# B&R Automation Studio project Y4_V3_1 (part 8)

#### S_Page13.st - Cyclic code
```iecst
(********************************************************************
 * COPYRIGHT --
 ********************************************************************
 * Program: S_Page13
 * File: S_Page13.st
 * Author: nicke
 * Created: May 02, 2013
 ********************************************************************
 * Implementation of program S_Page13
 ********************************************************************)

PROGRAM _CYCLIC

	//SETTINGS SCREEN
	ServiceVis.P13.EnableIndex	:=	LIMIT(0,ServiceVis.P13.EnableIndex,24)	;
	ServiceVis.P13.Status[0]	:=	HIDE	;
	ServiceVis.P13.Status[1]	:=	HIDE	;
	ServiceVis.P13.Status[2]	:=	HIDE	;
	ServiceVis.P13.Status[3]	:=	HIDE	;
	ServiceVis.P13.Status[4]	:=	HIDE	;
	ServiceVis.P13.Status[5]	:=	HIDE	;
	ServiceVis.P13.Status[6]	:=	HIDE	;
	ServiceVis.P13.Status[7]	:=	HIDE	;
	ServiceVis.P13.Status[8]	:=	HIDE	;
	ServiceVis.P13.Status[9]	:=	HIDE	;
	ServiceVis.P13.Status[10]	:=	HIDE	;
	ServiceVis.P13.Colour[1]	:=	BLUE	;
	ServiceVis.P13.Colour[2]	:=	BLUE	;
	ServiceVis.P13.Colour[3]	:=	BLUE	;
	ServiceVis.P13.Colour[4]	:=	BLUE	;
	ServiceVis.P13.Colour[5]	:=	BLUE	;
	ServiceVis.P13.Colour[6]	:=	BLUE	;

	CASE ServiceVis.P13.EnableIndex OF
		0:
			ServiceVis.P13.Status[0]	:=	SHOW	;
			ServiceVis.CalcBelt.Disp	:=	HIDE	;
		1:
			ServiceVis.P13.Status[1]	:=	SHOW	;
			ServiceVis.P13.Status[9]	:=	SHOW	;
			ServiceVis.P13.Colour[1]	:=	BLUE_ACTIVE	;
		2:
			ServiceVis.P13.Status[2]	:=	SHOW	;
			ServiceVis.P13.Status[9]	:=	SHOW	;
			ServiceVis.P13.Colour[2]	:=	BLUE_ACTIVE	;
			ServiceVis.CalcBelt.Disp	:=	HIDE	;
		3:
			ServiceVis.P13.Status[3]	:=	SHOW	;
			ServiceVis.P13.Status[9]	:=	SHOW	;
			ServiceVis.P13.Colour[3]	:=	BLUE_ACTIVE	;
			ServiceVis.CalcBelt.Disp	:=	HIDE	;
		4:
			ServiceVis.P13.Status[4]	:=	SHOW	;
			ServiceVis.P13.Status[9]	:=	SHOW	;
			ServiceVis.P13.Colour[4]	:=	BLUE_ACTIVE	;
			ServiceVis.CalcBelt.Disp	:=	HIDE	;
		5:
			ServiceVis.P13.Status[5]	:=	SHOW	;
			ServiceVis.P13.Status[9]	:=	SHOW	;
			ServiceVis.P13.Colour[5]	:=	BLUE_ACTIVE	;
			ServiceVis.CalcBelt.Disp	:=	HIDE	;
		6:
			ServiceVis.P13.Status[6]	:=	SHOW	;
			ServiceVis.P13.Status[9]	:=	SHOW	;
			ServiceVis.P13.Colour[6]	:=	BLUE_ACTIVE	;
			ServiceVis.CalcBelt.Disp	:=	HIDE	;
		7:
			ServiceVis.P13.Status[7]	:=	SHOW	;
			ServiceVis.CalcBelt.Disp	:=	HIDE	;
		8:
			ServiceVis.P13.Status[8]	:=	SHOW	;
			ServiceVis.P13.Status[3]	:=	SHOW	;
			ServiceVis.P13.Status[9]	:=	SHOW	;
			ServiceVis.P13.Colour[3]	:=	BLUE_ACTIVE	;
			ServiceVis.CalcBelt.Disp	:=	HIDE	;
		10:
			ServiceVis.P13.Status[10]	:=	SHOW	;
			ServiceVis.P13.Status[6]	:=	SHOW	;
			ServiceVis.P13.Status[9]	:=	SHOW	;
			ServiceVis.P13.Colour[6]	:=	BLUE_ACTIVE	;
			ServiceVis.CalcBelt.Disp	:=	HIDE	;

	END_CASE

	//CALCULATE WHEN LAYER HAS CHANGED
	ServiceVis.P13.Changed	:=	FALSE	;
	ServiceVis.P13.New	:=	ServiceVis.P13.EnableIndex	;
	IF(ServiceVis.P13.New <> ServiceVis.P13.Old) THEN
		ServiceVis.P13.Changed	:=	TRUE	;
	END_IF
	IF EDGEPOS(ServiceVis.P13.Changed) THEN
		ServiceVis.P13Delays.EnableIndex	:=	24	;
		ServiceVis.P13Servos.EnableIndex	:=	24	;
		ServiceVis.P13System.EnableIndex	:=	24	;
		ServiceVis.P13Timeouts.EnableIndex	:=	24	;
		ServiceVis.P13Help1.EnableIndex	:=	24	;
		ServiceVis.P13Help2.EnableIndex	:=	24	;
	END_IF
	ServiceVis.P13.Old	:=	ServiceVis.P13.EnableIndex	;

	//SETTINGS DELAYS SCREEN
	ServiceVis.P13Delays.Status[0]	:=	HIDE	;
	ServiceVis.P13Delays.Status[1]	:=	HIDE	;
	ServiceVis.P13Delays.Status[2]	:=	HIDE	;
	ServiceVis.P13Delays.Status[3]	:=	HIDE	;
	ServiceVis.P13Delays.Status[4]	:=	HIDE	;
	ServiceVis.P13Delays.Status[5]	:=	HIDE	;
	ServiceVis.P13Delays.Status[6]	:=	HIDE	;
	ServiceVis.P13Delays.Status[7]	:=	HIDE	;
	ServiceVis.P13Delays.Status[8]	:=	HIDE	;
	ServiceVis.P13Delays.Status[9]	:=	HIDE	;
	ServiceVis.P13Delays.Status[10]	:=	HIDE	;
	ServiceVis.P13Delays.Colour[0]	:=	BLUE	;
	ServiceVis.P13Delays.Colour[1]	:=	BLUE	;
	ServiceVis.P13Delays.Colour[2]	:=	BLUE	;
	ServiceVis.P13Delays.Colour[3]	:=	BLUE	;
	ServiceVis.P13Delays.Colour[4]	:=	BLUE	;
	ServiceVis.P13Delays.Colour[5]	:=	BLUE	;
	ServiceVis.P13Delays.Colour[6]	:=	BLUE	;
	ServiceVis.P13Delays.Colour[7]	:=	BLUE	;
	ServiceVis.P13Delays.Colour[8]	:=	BLUE	;

	CASE ServiceVis.P13Delays.EnableIndex OF
		0..8://LayerDelay[1..9]
			ServiceVis.P13Delays.Status[ServiceVis.P13Delays.EnableIndex]	:=	SHOW	;
			ServiceVis.P13Delays.Colour[ServiceVis.P13Delays.EnableIndex]	:=	BLUE_ACTIVE	;
			ServiceVis.P13Delays.Status[9]	:=	SHOW	;//LayerDelays
			ServiceVis.P13.Status[1]	:=	HIDE	;//Layer2
			ServiceVis.P13.Status[9]	:=	HIDE	;//Layers
		10:
			ServiceVis.P13Delays.Status[10]	:=	SHOW	;
	END_CASE

	CASE ServiceVis.P13Delays.EnableIndex OF
		0,2,4,5,6,7,8,24:
			ServiceVis.CalcBelt.Disp	:=	HIDE	;
	END_CASE

	//CALCULATE WHEN LAYER HAS CHANGED
	ServiceVis.P13Delays.Changed	:=	FALSE	;
	ServiceVis.P13Delays.New	:=	ServiceVis.P13Delays.EnableIndex	;
	IF(ServiceVis.P13Delays.New <> ServiceVis.P13Delays.Old) THEN
		ServiceVis.P13Delays.Changed	:=	TRUE	;
	END_IF
	IF EDGEPOS(ServiceVis.P13Delays.Changed) THEN
		ServiceVis.P13Help1.EnableIndex	:=	24	;
		ServiceVis.P13Help2.EnableIndex	:=	24	;
	END_IF
	ServiceVis.P13Delays.Old	:=	ServiceVis.P13Delays.EnableIndex	;

	//CALCULATOR FOR BELT DISPLAY
	IF (ServiceVis.CalcBelt.Disp = SHOW) THEN
		IF (ServiceVis.CalcBelt.Delay) THEN
			ServiceVis.CalcBelt.Adjust	:= 	1 - ((ServiceVis.CalcBelt.Unground + 300)/(Speeds.SpeedSeam/6))	;
		ELSE
			ServiceVis.CalcBelt.Adjust	:= 	(ServiceVis.CalcBelt.Unground + 300)/(Speeds.SpeedSeam/6);
		END_IF
		ServiceVis.CalcBelt.New	:= 	(ServiceVis.CalcBelt.Current + ServiceVis.CalcBelt.Adjust)	;

		IF (ServiceVis.CalcBelt.Unground = 0) THEN
			ServiceVis.CalcBelt.Adjust	:= 	0	;
			ServiceVis.CalcBelt.New	:= 	0	;
		END_IF
	END_IF

	//SETTINGS DRIVES SCREEN
	ServiceVis.P13Drives.Status[0]	:=	HIDE	;
	ServiceVis.P13Drives.Status[1]	:=	HIDE	;
	ServiceVis.P13Drives.Status[2]	:=	HIDE	;
	ServiceVis.P13Drives.Status[3]	:=	HIDE	;
	ServiceVis.P13Drives.Status[4]	:=	HIDE	;
	ServiceVis.P13Drives.Status[5]	:=	HIDE	;
	ServiceVis.P13Drives.Status[6]	:=	HIDE	;
	ServiceVis.P13Drives.Status[7]	:=	HIDE	;
	ServiceVis.P13Drives.Status[8]	:=	HIDE	;
	ServiceVis.P13Drives.Status[9]	:=	HIDE	;
	ServiceVis.P13Drives.Status[10]:=	HIDE	;
	ServiceVis.P13Drives.Status[11]:=	HIDE	;
	ServiceVis.P13Drives.Status[12]:=	HIDE	;
	ServiceVis.P13Drives.Status[13]:=	HIDE	;
	ServiceVis.P13Drives.Status[14]:=	HIDE	;
	ServiceVis.P13Drives.Status[15]:=	HIDE	;
	ServiceVis.P13Drives.Status[20]:=	HIDE	;
	ServiceVis.P13Drives.Status[21]:=	HIDE	;
	ServiceVis.P13Drives.Status[22]:=	HIDE	;
	ServiceVis.P13Drives.Colour[0]	:=	BLUE	;
	ServiceVis.P13Drives.Colour[1]	:=	BLUE	;
	ServiceVis.P13Drives.Colour[2]	:=	BLUE	;
	ServiceVis.P13Drives.Colour[3]	:=	BLUE	;
	ServiceVis.P13Drives.Colour[4]	:=	BLUE	;
	ServiceVis.P13Drives.Colour[5]	:=	BLUE	;
	ServiceVis.P13Drives.Colour[6]	:=	BLUE	;

	CASE ServiceVis.P13Drives.EnableIndex OF
		0..6:
			ServiceVis.P13Drives.Status[ServiceVis.P13Drives.EnableIndex]	:=	SHOW	;
			ServiceVis.P13Drives.Colour[ServiceVis.P13Drives.EnableIndex]	:=	BLUE_ACTIVE	;
			ServiceVis.P13Drives.Status[9]	:=	SHOW	;
			ServiceVis.P13.Status[2]	:=	HIDE	;
			ServiceVis.P13.Status[9]	:=	HIDE	;
			IF(ServiceLevel.Level > SUPERVISOR) THEN
				ServiceVis.P13Drives.Status[ServiceVis.P13Drives.EnableIndex + 9]	:=	SHOW	;
			END_IF
		7:
			ServiceVis.P13Drives.Status[7]	:=	SHOW	;
		8:
			ServiceVis.P13Drives.Status[8]	:=	SHOW	;
	END_CASE

	//CALCULATE WHEN LAYER HAS CHANGED
	ServiceVis.P13Drives.Changed	:=	FALSE	;
	ServiceVis.P13Drives.New	:=	ServiceVis.P13Drives.EnableIndex	;
	IF(ServiceVis.P13Drives.New <> ServiceVis.P13Drives.Old) THEN
		ServiceVis.P13Drives.Changed	:=	TRUE	;
	END_IF
	IF EDGEPOS(ServiceVis.P13Drives.Changed) THEN
		ServiceVis.P13Help1.EnableIndex	:=	24	;
		ServiceVis.P13Help2.EnableIndex	:=	24	;
	END_IF
	ServiceVis.P13Drives.Old	:=	ServiceVis.P13Drives.EnableIndex	;

	//HIGHLIGHT SELECTED BATCHING MODE COLOUR
	CASE InvPerms.CLB.Analog OF
		NO_ANALOG:
			ServiceVis.P13.Colour[7]	:=	WHITE			;
			ServiceVis.P13.Colour[8]	:=	DROP_UNSELECTED	;
			ServiceVis.P13.Colour[9]	:=	DROP_UNSELECTED	;
			ServiceVis.P13.Colour[10]	:=	DROP_UNSELECTED	;
			ServiceVis.P13.Colour[11]	:=	DROP_UNSELECTED	;
		VOLTAGE_TYPE_1:
			ServiceVis.P13.Colour[7]	:=	DROP_UNSELECTED	;
			ServiceVis.P13.Colour[8]	:=	WHITE			;
			ServiceVis.P13.Colour[9]	:=	DROP_UNSELECTED	;
			ServiceVis.P13.Colour[10]	:=	DROP_UNSELECTED	;
			ServiceVis.P13.Colour[11]	:=	DROP_UNSELECTED	;
		CURRENT_TYPE_1:
			ServiceVis.P13.Colour[7]	:=	DROP_UNSELECTED	;
			ServiceVis.P13.Colour[8]	:=	DROP_UNSELECTED	;
			ServiceVis.P13.Colour[9]	:=	DROP_UNSELECTED	;
			ServiceVis.P13.Colour[10]	:=	WHITE			;
			ServiceVis.P13.Colour[11]	:=	DROP_UNSELECTED	;
		CURRENT_TYPE_2:
			ServiceVis.P13.Colour[7]	:=	DROP_UNSELECTED	;
			ServiceVis.P13.Colour[8]	:=	DROP_UNSELECTED	;
			ServiceVis.P13.Colour[9]	:=	DROP_UNSELECTED	;
			ServiceVis.P13.Colour[10]	:=	DROP_UNSELECTED	;
			ServiceVis.P13.Colour[11]	:=	WHITE			;
	END_CASE

	//SETTINGS SERVOS SCREEN
	ServiceVis.P13Servos.Status[0]	:=	HIDE	;
	ServiceVis.P13Servos.Status[1]	:=	HIDE	;
	ServiceVis.P13Servos.Status[2]	:=	HIDE	;
	ServiceVis.P13Servos.Status[3]	:=	HIDE	;
	ServiceVis.P13Servos.Status[4]	:=	HIDE	;
	ServiceVis.P13Servos.Status[5]	:=	HIDE	;
	ServiceVis.P13Servos.Status[6]	:=	HIDE	;
	ServiceVis.P13Servos.Status[7]	:=	HIDE	;
	ServiceVis.P13Servos.Status[8]	:=	HIDE	;
	ServiceVis.P13Servos.Status[9]	:=	HIDE	;
	ServiceVis.P13Servos.Colour[0]	:=	BLUE	;
	ServiceVis.P13Servos.Colour[1]	:=	BLUE	;
	ServiceVis.P13Servos.Colour[2]	:=	BLUE	;
	ServiceVis.P13Servos.Colour[3]	:=	BLUE	;
	ServiceVis.P13Servos.Colour[4]	:=	BLUE	;
	ServiceVis.P13Servos.Colour[5]	:=	BLUE	;
	ServiceVis.P13Servos.Colour[6]	:=	BLUE	;

	CASE ServiceVis.P13Servos.EnableIndex OF
		0..6:
			ServiceVis.P13Servos.Status[ServiceVis.P13Servos.EnableIndex]	:=	SHOW	;
			ServiceVis.P13Servos.Colour[ServiceVis.P13Servos.EnableIndex]	:=	BLUE_ACTIVE	;
			ServiceVis.P13Servos.Status[9]	:=	SHOW	;
			ServiceVis.P13.Status[2]	:=	HIDE	;
			ServiceVis.P13.Status[9]	:=	HIDE	;
		7:
			ServiceVis.P13Servos.Status[7]	:=	SHOW	;
		8:
			ServiceVis.P13Servos.Status[8]	:=	SHOW	;
	END_CASE

	//CALCULATE WHEN LAYER HAS CHANGED
	ServiceVis.P13Servos.Changed	:=	FALSE	;
	ServiceVis.P13Servos.New	:=	ServiceVis.P13Servos.EnableIndex	;
	IF(ServiceVis.P13Servos.New <> ServiceVis.P13Servos.Old) THEN
		ServiceVis.P13Servos.Changed	:=	TRUE	;
	END_IF
	IF EDGEPOS(ServiceVis.P13Servos.Changed) THEN
		ServiceVis.P13Help1.EnableIndex	:=	24	;
		ServiceVis.P13Help2.EnableIndex	:=	24	;
	END_IF
	ServiceVis.P13Servos.Old	:=	ServiceVis.P13Servos.EnableIndex	;

	//SETTINGS SYSTEM SCREEN
	ServiceVis.P13System.Status[0]	:=	HIDE	;
	ServiceVis.P13System.Status[1]	:=	HIDE	;
	ServiceVis.P13System.Status[2]	:=	HIDE	;
	ServiceVis.P13System.Status[3]	:=	HIDE	;
	ServiceVis.P13System.Status[4]	:=	HIDE	;
	ServiceVis.P13System.Status[5]	:=	HIDE	;
	ServiceVis.P13System.Status[6]	:=	HIDE	;
	ServiceVis.P13System.Status[7]	:=	HIDE	;
	ServiceVis.P13System.Status[8]	:=	HIDE	;
	ServiceVis.P13System.Status[9]	:=	HIDE	;
	ServiceVis.P13System.Colour[0]	:=	BLUE	;
	ServiceVis.P13System.Colour[1]	:=	BLUE	;
	ServiceVis.P13System.Colour[2]	:=	BLUE	;
	ServiceVis.P13System.Colour[3]	:=	BLUE	;
	ServiceVis.P13System.Colour[4]	:=	BLUE	;
	ServiceVis.P13System.Colour[5]	:=	BLUE	;
	ServiceVis.P13System.Colour[6]	:=	BLUE	;

	CASE ServiceVis.P13System.EnableIndex OF
		0..6:
			ServiceVis.P13System.Status[ServiceVis.P13System.EnableIndex]	:=	SHOW	;
			ServiceVis.P13System.Colour[ServiceVis.P13System.EnableIndex]	:=	BLUE_ACTIVE	;
			ServiceVis.P13System.Status[9]	:=	SHOW	;
			ServiceVis.P13.Status[4]	:=	HIDE	;
			ServiceVis.P13.Status[9]	:=	HIDE	;
		7:
			ServiceVis.P13System.Status[7]	:=	SHOW	;
		8:
			ServiceVis.P13System.Status[8]	:=	SHOW	;
	END_CASE

	//CALCULATE WHEN LAYER HAS CHANGED
	ServiceVis.P13System.Changed	:=	FALSE	;
	ServiceVis.P13System.New	:=	ServiceVis.P13System.EnableIndex	;
	IF(ServiceVis.P13System.New <> ServiceVis.P13System.Old) THEN
		ServiceVis.P13System.Changed	:=	TRUE	;
	END_IF
	IF EDGEPOS(ServiceVis.P13System.Changed) THEN
		ServiceVis.P13Help1.EnableIndex	:=	24	;
		ServiceVis.P13Help2.EnableIndex	:=	24	;
	END_IF
	ServiceVis.P13System.Old	:=	ServiceVis.P13System.EnableIndex	;

	//SETTINGS TIMEOUT SCREEN
	ServiceVis.P13Timeouts.Status[0]	:=	HIDE	;
	ServiceVis.P13Timeouts.Status[1]	:=	HIDE	;
	ServiceVis.P13Timeouts.Status[2]	:=	HIDE	;
	ServiceVis.P13Timeouts.Status[3]	:=	HIDE	;
	ServiceVis.P13Timeouts.Status[4]	:=	HIDE	;
	ServiceVis.P13Timeouts.Status[5]	:=	HIDE	;
	ServiceVis.P13Timeouts.Status[6]	:=	HIDE	;
	ServiceVis.P13Timeouts.Status[7]	:=	HIDE	;
	ServiceVis.P13Timeouts.Status[8]	:=	HIDE	;
	ServiceVis.P13Timeouts.Status[9]	:=	HIDE	;
	ServiceVis.P13Timeouts.Colour[0]	:=	BLUE	;
	ServiceVis.P13Timeouts.Colour[1]	:=	BLUE	;
	ServiceVis.P13Timeouts.Colour[2]	:=	BLUE	;
	ServiceVis.P13Timeouts.Colour[3]	:=	BLUE	;
	ServiceVis.P13Timeouts.Colour[4]	:=	BLUE	;
	ServiceVis.P13Timeouts.Colour[5]	:=	BLUE	;
	ServiceVis.P13Timeouts.Colour[6]	:=	BLUE	;

	CASE ServiceVis.P13Timeouts.EnableIndex OF
		0..6:
			ServiceVis.P13Timeouts.Status[ServiceVis.P13Timeouts.EnableIndex]	:=	SHOW	;
			ServiceVis.P13Timeouts.Colour[ServiceVis.P13Timeouts.EnableIndex]	:=	BLUE_ACTIVE	;
			ServiceVis.P13Timeouts.Status[9]	:=	SHOW	;
			ServiceVis.P13.Status[5]	:=	HIDE	;
			ServiceVis.P13.Status[9]	:=	HIDE	;
		7:
			ServiceVis.P13Timeouts.Status[7]	:=	SHOW	;
		8:
			ServiceVis.P13Timeouts.Status[8]	:=	SHOW	;
	END_CASE

	//CALCULATE WHEN LAYER HAS CHANGED
	ServiceVis.P13Timeouts.Changed	:=	FALSE	;
	ServiceVis.P13Timeouts.New	:=	ServiceVis.P13Timeouts.EnableIndex	;
	IF(ServiceVis.P13Timeouts.New <> ServiceVis.P13Timeouts.Old) THEN
		ServiceVis.P13Timeouts.Changed	:=	TRUE	;
	END_IF
	IF EDGEPOS(ServiceVis.P13Timeouts.Changed) THEN
		ServiceVis.P13Help1.EnableIndex	:=	24	;
		ServiceVis.P13Help2.EnableIndex	:=	24	;
	END_IF
	ServiceVis.P13Timeouts.Old	:=	ServiceVis.P13Timeouts.EnableIndex	;

	//HELP LAYERS CONTROL
	memcpy(ADR(ServiceVis.P13Help1.Status),ADR(ServiceVis.HideAll),SIZEOF(ServiceVis.HideAll));
	ServiceVis.P13Help1.Colour[0]	:=	BLUE	;
	ServiceVis.P13Help1.Colour[1]	:=	BLUE	;
	ServiceVis.P13Help1.Colour[2]	:=	BLUE	;
	ServiceVis.P13Help1.Colour[3]	:=	BLUE	;
	ServiceVis.P13Help1.Colour[4]	:=	BLUE	;
	ServiceVis.P13Help1.Colour[5]	:=	BLUE	;
	ServiceVis.P13Help1.Colour[6]	:=	BLUE	;
	ServiceVis.P13Help1.Colour[7]	:=	BLUE	;
	ServiceVis.P13Help1.Colour[8]	:=	BLUE	;
	ServiceVis.P13Help1.Colour[9]	:=	BLUE	;

	CASE ServiceVis.P13Help1.EnableIndex OF
		0..23:
			ServiceVis.P13Help1.Status[ServiceVis.P13Help1.EnableIndex]	:=	SHOW	;
		24:
			ServiceVis.P13Help1.Index	:=	0	;
	END_CASE

	CASE ServiceVis.P13Help1.Index OF
		0..9:
			ServiceVis.P13Help1.Colour[ServiceVis.P13Help1.Index]	:=	BLUE_ACTIVE	;
	END_CASE

	//HELP LAYERS CONTROL 2
	memcpy(ADR(ServiceVis.P13Help2.Status),ADR(ServiceVis.HideAll),SIZEOF(ServiceVis.HideAll));
	ServiceVis.P13Help2.Colour[0]	:=	BLUE	;
	ServiceVis.P13Help2.Colour[1]	:=	BLUE	;
	ServiceVis.P13Help2.Colour[2]	:=	BLUE	;
	ServiceVis.P13Help2.Colour[3]	:=	BLUE	;
	ServiceVis.P13Help2.Colour[4]	:=	BLUE	;
	ServiceVis.P13Help2.Colour[5]	:=	BLUE	;
	ServiceVis.P13Help2.Colour[6]	:=	BLUE	;
	ServiceVis.P13Help2.Colour[7]	:=	BLUE	;
	ServiceVis.P13Help2.Colour[8]	:=	BLUE	;
	ServiceVis.P13Help2.Colour[9]	:=	BLUE	;
	ServiceVis.P13Help2.Colour[10]	:=	BLUE	;

	CASE ServiceVis.P13Help2.EnableIndex OF
		0..23:
			ServiceVis.P13Help2.Status[ServiceVis.P13Help2.EnableIndex]	:=	SHOW	;
		24:
			ServiceVis.P13Help2.Index	:=	0	;
	END_CASE

	CASE ServiceVis.P13Help2.Index OF
		0..10:
			ServiceVis.P13Help2.Colour[ServiceVis.P13Help2.Index]	:=	BLUE_ACTIVE	;
	END_CASE

END_PROGRAM
```

### Program Logical/VisControl/ServiceControl/S_Page14 (IEC) - Drives screen control

#### S_Page14.st - Cyclic code
```iecst
(********************************************************************
 * COPYRIGHT --
 ********************************************************************
 * Program: S_Page14
 * File: S_Page14.st
 * Author: nicke
 * Created: May 02, 2013
 ********************************************************************
 * Implementation of program S_Page14
 ********************************************************************)

PROGRAM _CYCLIC

	//DRIVES SCREEN
	memcpy(ADR(ServiceVis.P14.Status),ADR(ServiceVis.HideAll),SIZEOF(ServiceVis.HideAll));
	ServiceVis.P14.Colour[0]	:=	VIOLET	;
	ServiceVis.P14.Colour[1]	:=	VIOLET	;
	ServiceVis.P14.Colour[2]	:=	VIOLET	;
	ServiceVis.P14.Colour[3]	:=	VIOLET	;
	ServiceVis.P14.Colour[4]	:=	VIOLET	;
	ServiceVis.P14.Colour[5]	:=	VIOLET	;
	ServiceVis.P14.Colour[6]	:=	VIOLET	;

	CASE ServiceVis.P14.EnableIndex OF
		0..6:
			ServiceVis.P14.Status[ServiceVis.P14.EnableIndex]	:=	SHOW	;
			ServiceVis.P14.Colour[ServiceVis.P14.EnableIndex]	:=	VIOLET_ACTIVE	;
	END_CASE

	IF (Control.Achieved1) OR(Control.Test) THEN
		ServiceVis.P14.Status[8]	:=	SHOW	;
	END_IF

	IF(Control.Test) THEN
		ServiceVis.P14.Status[9]	:=	SHOW	;
	END_IF

	//CALCULATE WHEN LAYER HAS CHANGED
	ServiceVis.P14.Changed	:=	FALSE	;
	ServiceVis.P14.New	:=	ServiceVis.P14.EnableIndex	;
	IF(ServiceVis.P14.New <> ServiceVis.P14.Old) THEN
		ServiceVis.P14.Changed	:=	TRUE	;
	END_IF
	IF EDGEPOS(ServiceVis.P14.Changed) THEN
		ServiceVis.P14Layer.EnableIndex		:=	24	;
		ServiceVis.P14Status.EnableIndex	:=	24	;
		ServiceVis.P14Help.EnableIndex		:=	24	;
	END_IF
	ServiceVis.P14.Old	:=	ServiceVis.P14.EnableIndex	;

	memcpy(ADR(ServiceVis.P14Layer.Status),ADR(ServiceVis.HideAll),SIZEOF(ServiceVis.HideAll));

	CASE ServiceVis.P14Layer.EnableIndex OF
		0..19:
			ServiceVis.P14Layer.Status[ServiceVis.P14Layer.EnableIndex]	:=	SHOW	;
	END_CASE

END_PROGRAM
```

### Program Logical/VisControl/ServiceControl/S_Page15 (IEC) - Servo screen control

#### S_Page15.st - Cyclic code
```iecst
(********************************************************************
 * COPYRIGHT --
 ********************************************************************
 * Program: S_Page15
 * File: S_Page15.st
 * Author: nicke
 * Created: May 02, 2013
 ********************************************************************
 * Implementation of program S_Page15
 ********************************************************************)

PROGRAM _CYCLIC

	//SERVOS SCREEN
	memcpy(ADR(ServiceVis.P15.Status),ADR(ServiceVis.HideAll),SIZEOF(ServiceVis.HideAll));
	ServiceVis.P15.Colour[0]	:=	GREEN1	;
	ServiceVis.P15.Colour[1]	:=	GREEN1	;
	ServiceVis.P15.Colour[2]	:=	GREEN1	;
	ServiceVis.P15.Colour[3]	:=	GREEN1	;
	ServiceVis.P15.Colour[4]	:=	GREEN1	;
	ServiceVis.P15.Colour[5]	:=	GREEN1	;
	ServiceVis.P15.Colour[6]	:=	GREEN1	;

	CASE ServiceVis.P15.EnableIndex OF
		0..6:
			ServiceVis.P15.Status[ServiceVis.P15.EnableIndex]	:=	SHOW	;
			ServiceVis.P15.Colour[ServiceVis.P15.EnableIndex]	:=	GREEN1_ACTIVE	;
	END_CASE

	IF(Control.Test) THEN
		ServiceVis.P15.Status[8]	:=	SHOW	;
		//	ELSE
		//		ServiceVis.P15Layer.EnableIndex	:=	24	;
	END_IF

	//CALCULATE WHEN LAYER HAS CHANGED
	ServiceVis.P15.Changed	:=	FALSE	;
	ServiceVis.P15.New	:=	ServiceVis.P15.EnableIndex	;
	IF(ServiceVis.P15.New <> ServiceVis.P15.Old) THEN
		ServiceVis.P15.Changed	:=	TRUE	;
	END_IF
	IF EDGEPOS(ServiceVis.P15.Changed) THEN
		ServiceVis.P15Layer.EnableIndex	:=	24	;
	END_IF
	ServiceVis.P15.Old	:=	ServiceVis.P15.EnableIndex	;

	memcpy(ADR(ServiceVis.P15Layer.Status),ADR(ServiceVis.HideAll),SIZEOF(ServiceVis.HideAll));

	CASE ServiceVis.P15Layer.EnableIndex OF
		0..15:
			ServiceVis.P15Layer.Status[ServiceVis.P15Layer.EnableIndex]	:=	SHOW	;
	END_CASE

	IF(Control.Test) THEN
	ELSE
		ServiceVis.P15Layer.Status[0]	:=	HIDE	;
		ServiceVis.P15Layer.Status[1]	:=	HIDE	;
		ServiceVis.P15Layer.Status[2]	:=	HIDE	;
	END_IF

END_PROGRAM
```

### Program Logical/VisControl/ServiceControl/S_Page16 (IEC) - Remote screen control

#### S_Page16.st - Cyclic code
```iecst
(********************************************************************
 * COPYRIGHT --
 ********************************************************************
 * Program: S_Page16
 * File: S_Page16.st
 * Author: nicke
 * Created: May 02, 2013
 ********************************************************************
 * Implementation of program S_Page16
 ********************************************************************)

PROGRAM _CYCLIC

	//REMOTE SCREEN
	memcpy(ADR(ServiceVis.P16.Status),ADR(ServiceVis.HideAll),SIZEOF(ServiceVis.HideAll));
	ServiceVis.P16.Colour[0]	:=	LIGHTBLUE	;
	ServiceVis.P16.Colour[1]	:=	LIGHTBLUE	;
	ServiceVis.P16.Colour[2]	:=	LIGHTBLUE	;
	ServiceVis.P16.Colour[3]	:=	LIGHTBLUE	;
	ServiceVis.P16.Colour[4]	:=	LIGHTBLUE	;
	ServiceVis.P16.Colour[5]	:=	LIGHTBLUE	;
	ServiceVis.P16.Colour[6]	:=	LIGHTBLUE	;
	ServiceVis.P16.Colour[7]	:=	LIGHTBLUE	;
	ServiceVis.P16.Colour[8]	:=	LIGHTBLUE	;
	ServiceVis.P16.Colour[9]	:=	LIGHTBLUE	;
	ServiceVis.P16.Colour[10]	:=	LIGHTBLUE	;

	CASE ServiceVis.P16.EnableIndex OF
		0..7,9,10:
			ServiceVis.P16.Status[ServiceVis.P16.EnableIndex]	:=	SHOW	;
			ServiceVis.P16.Colour[ServiceVis.P16.EnableIndex]	:=	LIGHTBLUE_ACTIVE	;
	END_CASE

	IF(Control.Test) THEN
		ServiceVis.P16.Status[8]	:=	SHOW	;
	ELSE
		ServiceVis.P16.EnableIndex	:= LIMIT(0, ServiceVis.P16.EnableIndex, 6);
	END_IF

	//CALCULATE WHEN LAYER HAS CHANGED
	ServiceVis.P16.Changed	:=	FALSE	;
	ServiceVis.P16.New	:=	ServiceVis.P16.EnableIndex	;
	IF(ServiceVis.P16.New <> ServiceVis.P16.Old) THEN
		ServiceVis.P16.Changed	:=	TRUE	;
	END_IF
	IF EDGEPOS(ServiceVis.P16.Changed) THEN
		ServiceVis.P16Layer.EnableIndex	:=	24	;
	END_IF
	ServiceVis.P16.Old	:=	ServiceVis.P16.EnableIndex	;

	memcpy(ADR(ServiceVis.P16Layer.Status),ADR(ServiceVis.HideAll),SIZEOF(ServiceVis.HideAll));

	CASE ServiceVis.P16Layer.EnableIndex OF
		0..15:
			ServiceVis.P16Layer.Status[ServiceVis.P16Layer.EnableIndex]	:=	SHOW	;
	END_CASE

END_PROGRAM
```

### Program Logical/VisControl/ServiceControl/S_Page18 (IEC) - Warning screen control

#### S_Page18.st - Cyclic code
```iecst
(********************************************************************
 * COPYRIGHT --
 ********************************************************************
 * Program: S_Page18
 * File: S_Page18.st
 * Author: nicke
 * Created: May 02, 2013
 ********************************************************************
 * Implementation of program S_Page18
 ********************************************************************)

PROGRAM _CYCLIC

(* Section to control pop up warnings for flip arms *)
(*Seamer 1 Down *)
	ServiceVis.FlipDisp1.Runtime1	:=	HIDE	;
	ServiceVis.FlipDisp1.Runtime2	:=	HIDE	;
	ServiceVis.FlipDisp1.Runtime3	:=	HIDE	;
	ServiceVis.FlipDisp1.Runtime4	:=	HIDE	;

	IF ((Ax1.Active) OR NOT(Ax1.OriginSet)) AND NOT(Ax1.Block) AND(Control.Achieved1) THEN
		ServiceVis.FlipDisp1.Runtime1	:=	SHOW	;
		ServiceVis.FlipDisp1.TextIndex1	:=	BOOL_TO_USINT(NOT(S100Reed.In))	;
		ServiceVis.FlipDisp1.TextIndex2	:=	BOOL_TO_USINT(NOT(S102Reed.In))	;
		ServiceVis.FlipDisp1.TextIndex3	:=	BOOL_TO_USINT(NOT(S104Reed.In))	;
		ServiceVis.FlipDisp1.TextIndex4	:=	BOOL_TO_USINT(NOT(S106Reed.In))	;
		ServiceVis.FlipDisp1.TextIndex5	:=	BOOL_TO_USINT(NOT(S108Reed.In))	;
		ServiceVis.FlipDisp1.TextIndex6	:=	BOOL_TO_USINT(NOT(S110Reed.In))	;
		ServiceVis.FlipDisp1.TextIndex7	:=	BOOL_TO_USINT(NOT(S112Reed.In))	;
		ServiceVis.FlipDisp1.TextIndex8	:=	BOOL_TO_USINT(NOT(S114Reed.In))	;
		ServiceVis.FlipDisp1.TextIndex9	:=	BOOL_TO_USINT(NOT(S116Reed.In))	;
		ServiceVis.FlipDisp1.TextIndex10	:=	BOOL_TO_USINT(NOT(S118Reed.In))	;
		CASE Perms.FLIPARMS1 OF
			3:
				ServiceVis.FlipDisp1.Runtime2		:=	SHOW	;
			4:
				ServiceVis.FlipDisp1.Runtime2		:=	SHOW	;
				ServiceVis.FlipDisp1.Runtime3		:=	SHOW	;
			5:
				ServiceVis.FlipDisp1.Runtime2		:=	SHOW	;
				ServiceVis.FlipDisp1.Runtime3		:=	SHOW	;
				ServiceVis.FlipDisp1.Runtime4		:=	SHOW	;
		END_CASE
	END_IF

	(* Seamer 1 Up *)
	ServiceVis.FlipDisp1.Runtime5	:= HIDE	;
	ServiceVis.FlipDisp1.Runtime6	:= HIDE	;
	ServiceVis.FlipDisp1.Runtime7	:= HIDE	;
	ServiceVis.FlipDisp1.Runtime8	:= HIDE	;
	ServiceVis.FlipDisp1.Runtime9	:= HIDE	;
	ServiceVis.FlipDisp1.TextIndex11	:=	BOOL_TO_USINT(NOT(S101Reed.In))	;
	ServiceVis.FlipDisp1.TextIndex12	:=	BOOL_TO_USINT(NOT(S103Reed.In))	;
	ServiceVis.FlipDisp1.TextIndex13	:=	BOOL_TO_USINT(NOT(S105Reed.In))	;
	ServiceVis.FlipDisp1.TextIndex14	:=	BOOL_TO_USINT(NOT(S107Reed.In))	;
	ServiceVis.FlipDisp1.TextIndex15	:=	BOOL_TO_USINT(NOT(S109Reed.In))	;
	ServiceVis.FlipDisp1.TextIndex16	:=	BOOL_TO_USINT(NOT(S111Reed.In))	;
	ServiceVis.FlipDisp1.TextIndex17	:=	BOOL_TO_USINT(NOT(S113Reed.In))	;
	ServiceVis.FlipDisp1.TextIndex18	:=	BOOL_TO_USINT(NOT(S115Reed.In))	;
	ServiceVis.FlipDisp1.TextIndex19	:=	BOOL_TO_USINT(NOT(S117Reed.In))	;
	ServiceVis.FlipDisp1.TextIndex20	:=	BOOL_TO_USINT(NOT(S119Reed.In))	;
	CASE ArmsTemp2.CheckRaised OF
		0:	(* No arms up *)
		1:	(* 1 arm up *)
			ServiceVis.FlipDisp1.Runtime5	:= SHOW	;
		2:	(* 2 arms up *)
			ServiceVis.FlipDisp1.Runtime5	:= SHOW	;
			ServiceVis.FlipDisp1.Runtime6	:= SHOW	;
		3:  (* 3 arms up *)
			ServiceVis.FlipDisp1.Runtime5	:= SHOW	;
			ServiceVis.FlipDisp1.Runtime6	:= SHOW	;
			ServiceVis.FlipDisp1.Runtime7	:= SHOW	;
		4:	(* 4 arms up *)
			ServiceVis.FlipDisp1.Runtime5	:= SHOW	;
			ServiceVis.FlipDisp1.Runtime6	:= SHOW	;
			ServiceVis.FlipDisp1.Runtime7	:= SHOW	;
			ServiceVis.FlipDisp1.Runtime8	:= SHOW	;
		5:	(* 5 arms up *)
			ServiceVis.FlipDisp1.Runtime5	:= SHOW	;
			ServiceVis.FlipDisp1.Runtime6	:= SHOW	;
			ServiceVis.FlipDisp1.Runtime7	:= SHOW	;
			ServiceVis.FlipDisp1.Runtime8	:= SHOW	;
			ServiceVis.FlipDisp1.Runtime9	:= SHOW	;
	END_CASE

	(* Seamer 2 Down *)
	ServiceVis.FlipDisp2.Runtime1	:=	HIDE	;
	ServiceVis.FlipDisp2.Runtime2	:=	HIDE	;
	ServiceVis.FlipDisp2.Runtime3	:=	HIDE	;
	ServiceVis.FlipDisp2.Runtime4	:=	HIDE	;

	IF ((Ax2.Active) OR NOT(Ax2.OriginSet)) AND NOT(Ax2.Block) AND(Control.Achieved1) THEN
		ServiceVis.FlipDisp2.Runtime1	:=	SHOW	;
		ServiceVis.FlipDisp2.TextIndex1	:=	BOOL_TO_USINT(NOT(S120Reed.In))	;
		ServiceVis.FlipDisp2.TextIndex2	:=	BOOL_TO_USINT(NOT(S122Reed.In))	;
		ServiceVis.FlipDisp2.TextIndex3	:=	BOOL_TO_USINT(NOT(S124Reed.In))	;
		ServiceVis.FlipDisp2.TextIndex4	:=	BOOL_TO_USINT(NOT(S126Reed.In))	;
		ServiceVis.FlipDisp2.TextIndex5	:=	BOOL_TO_USINT(NOT(S128Reed.In))	;
		ServiceVis.FlipDisp2.TextIndex6	:=	BOOL_TO_USINT(NOT(S130Reed.In))	;
		ServiceVis.FlipDisp2.TextIndex7	:=	BOOL_TO_USINT(NOT(S132Reed.In))	;
		ServiceVis.FlipDisp2.TextIndex8	:=	BOOL_TO_USINT(NOT(S134Reed.In))	;
		ServiceVis.FlipDisp2.TextIndex9	:=	BOOL_TO_USINT(NOT(S136Reed.In))	;
		ServiceVis.FlipDisp2.TextIndex10	:=	BOOL_TO_USINT(NOT(S138Reed.In))	;
		CASE Perms.FLIPARMS2 OF
			3:
				ServiceVis.FlipDisp2.Runtime2	:=	SHOW	;
			4:
				ServiceVis.FlipDisp2.Runtime2	:=	SHOW	;
				ServiceVis.FlipDisp2.Runtime3	:=	SHOW	;
			5:
				ServiceVis.FlipDisp2.Runtime2	:=	SHOW	;
				ServiceVis.FlipDisp2.Runtime3	:=	SHOW	;
				ServiceVis.FlipDisp2.Runtime4	:=	SHOW	;
		END_CASE
	END_IF

	(* Seamer 2 Up *)
	ServiceVis.FlipDisp2.Runtime5	:= HIDE	;
	ServiceVis.FlipDisp2.Runtime6	:= HIDE	;
	ServiceVis.FlipDisp2.Runtime7	:= HIDE	;
	ServiceVis.FlipDisp2.Runtime8	:= HIDE	;
	ServiceVis.FlipDisp2.Runtime9	:= HIDE	;
	ServiceVis.FlipDisp2.TextIndex11	:=	BOOL_TO_USINT(NOT(S121Reed.In))	;
	ServiceVis.FlipDisp2.TextIndex12	:=	BOOL_TO_USINT(NOT(S123Reed.In))	;
	ServiceVis.FlipDisp2.TextIndex13	:=	BOOL_TO_USINT(NOT(S125Reed.In))	;
	ServiceVis.FlipDisp2.TextIndex14	:=	BOOL_TO_USINT(NOT(S127Reed.In))	;
	ServiceVis.FlipDisp2.TextIndex15	:=	BOOL_TO_USINT(NOT(S129Reed.In))	;
	ServiceVis.FlipDisp2.TextIndex16	:=	BOOL_TO_USINT(NOT(S131Reed.In))	;
	ServiceVis.FlipDisp2.TextIndex17	:=	BOOL_TO_USINT(NOT(S133Reed.In))	;
	ServiceVis.FlipDisp2.TextIndex18	:=	BOOL_TO_USINT(NOT(S135Reed.In))	;
	ServiceVis.FlipDisp2.TextIndex19	:=	BOOL_TO_USINT(NOT(S137Reed.In))	;
	ServiceVis.FlipDisp2.TextIndex20	:=	BOOL_TO_USINT(NOT(S139Reed.In))	;
	CASE ArmsTemp2.CheckRaised OF
		0:	(* No arms up *)
		1:	(* 1 arm up *)
			ServiceVis.FlipDisp2.Runtime5	:= SHOW	;
			ServiceVis.FlipDisp2.Runtime6	:= SHOW	;
		2:	(* 2 arms up *)
			ServiceVis.FlipDisp2.Runtime5	:= SHOW	;
			ServiceVis.FlipDisp2.Runtime6	:= SHOW	;
			ServiceVis.FlipDisp2.Runtime7	:= SHOW	;
		3:  (* 3 arms up *)
			ServiceVis.FlipDisp2.Runtime5	:= SHOW	;
			ServiceVis.FlipDisp2.Runtime6	:= SHOW	;
			ServiceVis.FlipDisp2.Runtime7	:= SHOW	;
			ServiceVis.FlipDisp2.Runtime8	:= SHOW	;
		4:	(* 4 arms up *)
			ServiceVis.FlipDisp2.Runtime5	:= SHOW	;
			ServiceVis.FlipDisp2.Runtime6	:= SHOW	;
			ServiceVis.FlipDisp2.Runtime7	:= SHOW	;
			ServiceVis.FlipDisp2.Runtime8	:= SHOW	;
			ServiceVis.FlipDisp2.Runtime9	:= SHOW	;
	END_CASE

END_PROGRAM
```

### Program Logical/VisControl/ServiceControl/S_Page20 (IEC) - Ashton tech screen control

#### S_Page20.st - Cyclic code
```iecst
(********************************************************************
 * COPYRIGHT --
 ********************************************************************
 * Program: S_Page20
 * File: S_Page20.st
 * Author: nicke
 * Created: May 02, 2013
 ********************************************************************
 * Implementation of program S_Page20
 ********************************************************************)

PROGRAM _CYCLIC

	//ASHTON TECH SCREEN
	memcpy(ADR(ServiceVis.P20.Status),ADR(ServiceVis.HideAll),SIZEOF(ServiceVis.HideAll));

	CASE ServiceVis.P20.EnableIndex OF
		0..7:
			ServiceVis.P20.Status[ServiceVis.P20.EnableIndex]	:=	SHOW	;
	END_CASE

END_PROGRAM
```

### Program Logical/VisControl/ServiceControl/S_ESRecover (IEC) - Estop recovery control

#### S_ESRecover.st - Cyclic code
```iecst
(********************************************************************
 * COPYRIGHT --
 ********************************************************************
 * Program: S_ESRecover
 * File: S_ESRecover.st
 * Author: nicke
 * Created: May 02, 2013
 ********************************************************************
 * Implementation of program S_ESRecover
 ********************************************************************)

PROGRAM _CYCLIC

(* Switch to EMO Recovery screen if any glass present *)
//	IF EDGEPOS(Control.EStop) AND (Control.Count > 0) THEN
//		ServiceVis.P11.EnableIndex	:= 	20	;
//		ServiceVis.Page.New	:=	P11_MIMIC	;
//	END_IF

	//ESTOP SCREEN CONTROL
	//??? ALWAYS ENSURE .EMO IS SET TO Vis. NOT ServiceVis.

END_PROGRAM
```

### Package Logical/HMIXGA - HMI Visualisation XGA Screens

- Visualisation Logical/HMIXGA/HMIXGA (not shown)

- Visualisation Logical/BatchDisplay/BatchP (not shown)

### Package Logical/InvComms - Handle comms to Inverters

### Program Logical/InvComms/EPLComms (IEC) - Program

#### EPLComms.typ - Local data types
```iecst
(********************************************************************
 * COPYRIGHT --
 ********************************************************************
 * Program: EPLComms
 * File: EPLComms.typ
 * Author: Bernecker + Rainer

 * Created: June 05, 2015
 ********************************************************************
 * Local data types of program epl
 ********************************************************************)

TYPE
	EPL_typ : 	STRUCT  (*Datatype for AsEPL Library*)
		Param : EPLParam_typ; (*Variable with Parameters*)
		FUB : EPLFUB_typ; (*Variable with Function Blocks*)
		State : EPLState_enum; (*State machine control variable*)
		INV : INVName_typ; (*Inverter Names*)
		ErrorCode : UDINT;
		Status : UDINT;
		Errorcount : USINT;
	END_STRUCT;
	EPLParam_typ : 	STRUCT  (*Datatype with parameters*)
		WriteData : UINT; (*Data to be written*)
	END_STRUCT;
	EPLFUB_typ : 	STRUCT  (*datatype with Function Blocks*)
		EPLWrite_0 : EplSDOWrite; (*FUB to write a node's object entries*)
	END_STRUCT;
	INVName_typ : 	STRUCT
		ACC : ARRAY[0..24]OF BOOL;
		ACCIndex : USINT;
		DEC : ARRAY[0..24]OF BOOL;
		DECIndex : USINT;
	END_STRUCT;
	EPLState_enum :
		(
		EPL_START := 0, (*State after system reboot*)
		EPL_INV1_ACCCHECK := 10, (*State to check if Acceleration ramp is changed*)
		EPL_INV1_ACCWRITE := 11, (*State to write Acceleration ramp*)
		EPL_INV1_DECCHECK := 12, (*State to check if Deceleration ramp is changed*)
		EPL_INV1_DECWRITE := 13, (*State to write Deceleration ramp*)
		EPL_INV2_ACCCHECK := 20, (*State to check if Acceleration ramp is changed*)
		EPL_INV2_ACCWRITE := 21, (*State to write Acceleration ramp*)
		EPL_INV2_DECCHECK := 22, (*State to check if Deceleration ramp is changed*)
		EPL_INV2_DECWRITE := 23, (*State to write Deceleration ramp*)
		EPL_INV3_ACCCHECK := 30, (*State to check if Acceleration ramp is changed*)
		EPL_INV3_ACCWRITE := 31, (*State to write Acceleration ramp*)
		EPL_INV3_DECCHECK := 32, (*State to check if Deceleration ramp is changed*)
		EPL_INV3_DECWRITE := 33, (*State to write Deceleration ramp*)
		EPL_INV4_ACCCHECK := 40, (*State to check if Acceleration ramp is changed*)
		EPL_INV4_ACCWRITE := 41, (*State to write Acceleration ramp*)
		EPL_INV4_DECCHECK := 42, (*State to check if Deceleration ramp is changed*)
		EPL_INV4_DECWRITE := 43, (*State to write Deceleration ramp*)
		EPL_INV5_ACCCHECK := 50, (*State to check if Acceleration ramp is changed*)
		EPL_INV5_ACCWRITE := 51, (*State to write Acceleration ramp*)
		EPL_INV5_DECCHECK := 52, (*State to check if Deceleration ramp is changed*)
		EPL_INV5_DECWRITE := 53, (*State to write Deceleration ramp*)
		EPL_INV6_ACCCHECK := 60, (*State to check if Acceleration ramp is changed*)
		EPL_INV6_ACCWRITE := 61, (*State to write Acceleration ramp*)
		EPL_INV6_DECCHECK := 62, (*State to check if Deceleration ramp is changed*)
		EPL_INV6_DECWRITE := 63, (*State to write Deceleration ramp*)
		EPL_INV7_ACCCHECK := 70, (*State to check if Acceleration ramp is changed*)
		EPL_INV7_ACCWRITE := 71, (*State to write Acceleration ramp*)
		EPL_INV7_DECCHECK := 72, (*State to check if Deceleration ramp is changed*)
		EPL_INV7_DECWRITE := 73, (*State to write Deceleration ramp*)
		EPL_INV8_ACCCHECK := 80, (*State to check if Acceleration ramp is changed*)
		EPL_INV8_ACCWRITE := 81, (*State to write Acceleration ramp*)
		EPL_INV8_DECCHECK := 82, (*State to check if Deceleration ramp is changed*)
		EPL_INV8_DECWRITE := 83, (*State to write Deceleration ramp*)
		EPL_INV9_ACCCHECK := 90, (*State to check if Acceleration ramp is changed*)
		EPL_INV9_ACCWRITE := 91, (*State to write Acceleration ramp*)
		EPL_INV9_DECCHECK := 92, (*State to check if Deceleration ramp is changed*)
		EPL_INV9_DECWRITE := 93, (*State to write Deceleration ramp*)
		EPL_INV10_ACCCHECK := 100, (*State to check if Acceleration ramp is changed*)
		EPL_INV10_ACCWRITE := 101, (*State to write Acceleration ramp*)
		EPL_INV10_DECCHECK := 102, (*State to check if Deceleration ramp is changed*)
		EPL_INV10_DECWRITE := 103, (*State to write Deceleration ramp*)
		EPL_INV11_ACCCHECK := 110, (*State to check if Acceleration ramp is changed*)
		EPL_INV11_ACCWRITE := 111, (*State to write Acceleration ramp*)
		EPL_INV11_DECCHECK := 112, (*State to check if Deceleration ramp is changed*)
		EPL_INV11_DECWRITE := 113, (*State to write Deceleration ramp*)
		EPL_INV12_ACCCHECK := 120, (*State to check if Acceleration ramp is changed*)
		EPL_INV12_ACCWRITE := 121, (*State to write Acceleration ramp*)
		EPL_INV12_DECCHECK := 122, (*State to check if Deceleration ramp is changed*)
		EPL_INV12_DECWRITE := 123, (*State to write Deceleration ramp*)
		EPL_INV13_ACCCHECK := 130, (*State to check if Acceleration ramp is changed*)
		EPL_INV13_ACCWRITE := 131, (*State to write Acceleration ramp*)
		EPL_INV13_DECCHECK := 132, (*State to check if Deceleration ramp is changed*)
		EPL_INV13_DECWRITE := 133, (*State to write Deceleration ramp*)
		EPL_INV14_ACCCHECK := 140, (*State to check if Acceleration ramp is changed*)
		EPL_INV14_ACCWRITE := 141, (*State to write Acceleration ramp*)
		EPL_INV14_DECCHECK := 142, (*State to check if Deceleration ramp is changed*)
		EPL_INV14_DECWRITE := 143, (*State to write Deceleration ramp*)
		EPL_INV15_ACCCHECK := 150, (*State to check if Acceleration ramp is changed*)
		EPL_INV15_ACCWRITE := 151, (*State to write Acceleration ramp*)
		EPL_INV15_DECCHECK := 152, (*State to check if Deceleration ramp is changed*)
		EPL_INV15_DECWRITE := 153, (*State to write Deceleration ramp*)
		EPL_INV16_ACCCHECK := 160, (*State to check if Acceleration ramp is changed*)
		EPL_INV16_ACCWRITE := 161, (*State to write Acceleration ramp*)
		EPL_INV16_DECCHECK := 162, (*State to check if Deceleration ramp is changed*)
		EPL_INV16_DECWRITE := 163, (*State to write Deceleration ramp*)
		EPL_INV17_ACCCHECK := 170, (*State to check if Acceleration ramp is changed*)
		EPL_INV17_ACCWRITE := 171, (*State to write Acceleration ramp*)
		EPL_INV17_DECCHECK := 172, (*State to check if Deceleration ramp is changed*)
		EPL_INV17_DECWRITE := 173, (*State to write Deceleration ramp*)
		EPL_INV18_ACCCHECK := 180, (*State to check if Acceleration ramp is changed*)
		EPL_INV18_ACCWRITE := 181, (*State to write Acceleration ramp*)
		EPL_INV18_DECCHECK := 182, (*State to check if Deceleration ramp is changed*)
		EPL_INV18_DECWRITE := 183, (*State to write Deceleration ramp*)
		EPL_INV19_ACCCHECK := 190, (*State to check if Acceleration ramp is changed*)
		EPL_INV19_ACCWRITE := 191, (*State to write Acceleration ramp*)
		EPL_INV19_DECCHECK := 192, (*State to check if Deceleration ramp is changed*)
		EPL_INV19_DECWRITE := 193, (*State to write Deceleration ramp*)
		EPL_INV20_ACCCHECK := 200, (*State to check if Acceleration ramp is changed*)
		EPL_INV20_ACCWRITE := 201, (*State to write Acceleration ramp*)
		EPL_INV20_DECCHECK := 202, (*State to check if Deceleration ramp is changed*)
		EPL_INV20_DECWRITE := 203, (*State to write Deceleration ramp*)
		EPL_INV21_ACCCHECK := 210, (*State to check if Acceleration ramp is changed*)
		EPL_INV21_ACCWRITE := 211, (*State to write Acceleration ramp*)
		EPL_INV21_DECCHECK := 212, (*State to check if Deceleration ramp is changed*)
		EPL_INV21_DECWRITE := 213, (*State to write Deceleration ramp*)
		EPL_INV22_ACCCHECK := 220, (*State to check if Acceleration ramp is changed*)
		EPL_WAIT := 240,
		EPL_ERROR := 250
		);
END_TYPE
```

#### EPLComms.var - Local variables
```iecst
(********************************************************************
 * COPYRIGHT --
 ********************************************************************
 * Program: EPLComms
 * File: EPL.var
 * Author: Bernecker + Rainer
 * Created: June 07, 2015
 ********************************************************************
 * Local variables of program EPL
 ********************************************************************)
VAR
	EPL : EPL_typ; (*Variable for the AsEPL Library*)
END_VAR
```

#### EPLComms.st - Implementation code
```iecst
(********************************************************************
 * COPYRIGHT --
 ********************************************************************
 * Program: EPLComms
 * File: EPLComms.st
 ********************************************************************
 * Implementation of program EPLComms
 ********************************************************************)

PROGRAM _INIT

	IF NOT(InvPerms.SetValues) THEN
		InvPerms.CL1.Accel  :=  5   ;
		InvPerms.CL1.Decel  :=  5   ;
		InvPerms.CS1.Accel  :=  5   ;
		InvPerms.CS1.Decel  :=  5   ;
		InvPerms.CV1.Accel  :=  5   ;
		InvPerms.CV1.Decel  :=  5   ;
		InvPerms.CC1.Accel  :=  5   ;
		InvPerms.CC1.Decel  :=  5   ;
		InvPerms.CC2.Accel  :=  5   ;
		InvPerms.CC2.Decel  :=  5   ;
		InvPerms.CS2.Accel  :=  5   ;
		InvPerms.CS2.Decel  :=  5   ;
		InvPerms.CV2.Accel  :=  5   ;
		InvPerms.CV2.Decel  :=  5   ;
		InvPerms.CC3.Accel  :=  5   ;
		InvPerms.CC3.Decel  :=  5   ;
		InvPerms.CC4.Accel  :=  5   ;
		InvPerms.CC4.Decel  :=  5   ;
		InvPerms.CB1.Accel  :=  5   ;
		InvPerms.CB1.Decel  :=  5   ;
		InvPerms.CB2.Accel  :=  5   ;
		InvPerms.CB2.Decel  :=  5   ;
		InvPerms.CRB.Accel  :=  5   ;
		InvPerms.CRB.Decel  :=  5   ;
		InvPerms.CRE.Accel  :=  5   ;
		InvPerms.CRE.Decel  :=  5   ;
		InvPerms.CLB.Accel  :=  5   ;
		InvPerms.CLB.Decel  :=  5   ;
		InvPerms.SetValues  :=  TRUE    ;
	END_IF

	EPL.State   :=  EPL_START   ;
	InvTemps    :=  InvPerms    ;

END_PROGRAM

PROGRAM _CYCLIC

    //SET LIMITS FOR ACCEL, 0.1 - 3 SECONDS
	InvTemps.CL1.Accel := LIMIT(1,InvTemps.CL1.Accel,30);
	InvTemps.CS1.Accel := LIMIT(1,InvTemps.CS1.Accel,30);
	InvTemps.CV1.Accel := LIMIT(1,InvTemps.CV1.Accel,30);
	InvTemps.CC1.Accel := LIMIT(1,InvTemps.CC1.Accel,30);
	InvTemps.CC2.Accel := LIMIT(1,InvTemps.CC2.Accel,30);
	InvTemps.CS2.Accel := LIMIT(1,InvTemps.CS2.Accel,30);
	InvTemps.CV2.Accel := LIMIT(1,InvTemps.CV2.Accel,30);
	InvTemps.CC3.Accel := LIMIT(1,InvTemps.CC3.Accel,30);
	InvTemps.CC4.Accel := LIMIT(1,InvTemps.CC4.Accel,30);
	InvTemps.CB1.Accel := LIMIT(1,InvTemps.CB1.Accel,30);
	InvTemps.CB2.Accel := LIMIT(1,InvTemps.CB2.Accel,30);
	InvTemps.CRB.Accel := LIMIT(1,InvTemps.CRB.Accel,30);
	InvTemps.CRE.Accel := LIMIT(1,InvTemps.CRE.Accel,30);
	InvTemps.CLB.Accel := LIMIT(1,InvTemps.CLB.Accel,30);
	//SET LIMITS FOR DECEL, 0.1 - 3 SECONDS
	InvTemps.CL1.Decel := LIMIT(1,InvTemps.CL1.Decel,30);
	InvTemps.CS1.Decel := LIMIT(1,InvTemps.CS1.Decel,30);
	InvTemps.CV1.Decel := LIMIT(1,InvTemps.CV1.Decel,30);
	InvTemps.CC1.Decel := LIMIT(1,InvTemps.CC1.Decel,30);
	InvTemps.CC2.Decel := LIMIT(1,InvTemps.CC2.Decel,30);
	InvTemps.CS2.Decel := LIMIT(1,InvTemps.CS2.Decel,30);
	InvTemps.CV2.Decel := LIMIT(1,InvTemps.CV2.Decel,30);
	InvTemps.CC3.Decel := LIMIT(1,InvTemps.CC3.Decel,30);
	InvTemps.CC4.Decel := LIMIT(1,InvTemps.CC4.Decel,30);
	InvTemps.CB1.Decel := LIMIT(1,InvTemps.CB1.Decel,30);
	InvTemps.CB2.Decel := LIMIT(1,InvTemps.CB2.Decel,30);
	InvTemps.CRB.Decel := LIMIT(1,InvTemps.CRB.Decel,30);
	InvTemps.CRE.Decel := LIMIT(1,InvTemps.CRE.Decel,30);
	InvTemps.CLB.Decel := LIMIT(1,InvTemps.CLB.Decel,30);

	CASE EPL.State OF
		EPL_START:
			IF(EPLState.LinkOK) THEN
				IF(EPLState.CycleOK) THEN
					IF(EPLState.SyncOK) THEN
						EPL.State   :=  EPL_INV1_ACCCHECK;
					END_IF
				END_IF
			END_IF

		EPL_INV1_ACCCHECK:
			IF(CL1.Module.OK) THEN
				IF(EPL.INV.ACC[1]) THEN
					IF(InvTemps.CL1.Accel <> InvPerms.CL1.Accel) THEN
						EPL.Param.WriteData := InvTemps.CL1.Accel;
						EPL.State := EPL_INV1_ACCWRITE;
					ELSE
						EPL.State := EPL_WAIT;
						EPL.INV.ACCIndex := 0;
					END_IF
				ELSE
					IF(InvPerms.CL1.Accel <> 5) THEN
						EPL.Param.WriteData := InvPerms.CL1.Accel;
						EPL.State := EPL_INV1_ACCWRITE;
					ELSE
						EPL.State := EPL_INV1_DECCHECK;
					END_IF
				END_IF
			END_IF

		EPL_INV1_ACCWRITE:

			EPL.FUB.EPLWrite_0.enable := 1;  //ENABLE FUB
			EPL.FUB.EPLWrite_0.pDevice := ADR('SL1.IF1.ST4');  //DEVICE NAME OF INVERTER
			EPL.FUB.EPLWrite_0.node := 4;  //NODE NUMBER OF THE STATION
			EPL.FUB.EPLWrite_0.index := 8252;  //WRITE INDEX 16#203C (DEC 8252)
			EPL.FUB.EPLWrite_0.subindex := 2;  //SUBINDEX #2 (DEC 2) : ACCELERATION RAMP
			EPL.FUB.EPLWrite_0.pData := ADR(EPL.Param.WriteData);  //POINTER TO THE DATA BEING WRITTEN
			EPL.FUB.EPLWrite_0.datalen := SIZEOF(EPL.Param.WriteData);  //SIZE OF THE DATA TO BE WRITTEN
			EPL.FUB.EPLWrite_0();

			IF EPL.FUB.EPLWrite_0.status = 0 THEN  //WRITE SUCCESSFUL
				EPL.FUB.EPLWrite_0.enable := 0;  //DISABLE THE FUB
				IF EPL.INV.ACC[1] THEN
					EPL.State := EPL_WAIT;
					EPL.INV.ACCIndex := 0;
					InvPerms.CL1.Accel := InvTemps.CL1.Accel;
				ELSE
					EPL.State := EPL_INV1_DECCHECK;
				END_IF
			ELSIF EPL.FUB.EPLWrite_0.status = ERR_FUB_BUSY THEN
				//BUSY
			ELSIF EPL.FUB.EPLWrite_0.status = ERR_FUB_ENABLE_FALSE THEN
				//DISABLED
			ELSE
				EPL.State := EPL_ERROR;
				EPL.INV.ACCIndex := 0;
			END_IF

		EPL_INV1_DECCHECK:
			IF(CL1.Module.OK) THEN
				IF(EPL.INV.DEC[1]) THEN
					IF(InvTemps.CL1.Decel <> InvPerms.CL1.Decel) THEN
						EPL.Param.WriteData := InvTemps.CL1.Decel;
						EPL.State := EPL_INV1_DECWRITE;
					ELSE
						EPL.State := EPL_WAIT;
						EPL.INV.DECIndex := 0;
					END_IF
				ELSE
					IF(InvPerms.CL1.Decel <> 5) THEN
						EPL.Param.WriteData := InvPerms.CL1.Decel;
						EPL.State := EPL_INV1_DECWRITE;
					ELSE
						EPL.State := EPL_INV2_ACCCHECK;
					END_IF
				END_IF
			END_IF

		EPL_INV1_DECWRITE:

			EPL.FUB.EPLWrite_0.enable := 1;  //ENABLE FUB
			EPL.FUB.EPLWrite_0.pDevice := ADR('SL1.IF1.ST4');  //DEVICE NAME OF INVERTER
			EPL.FUB.EPLWrite_0.node := 4;  //NODE NUMBER OF THE STATION
			EPL.FUB.EPLWrite_0.index := 8252;  //WRITE INDEX 16#203C (DEC 8252)
			EPL.FUB.EPLWrite_0.subindex := 3;  //SUBINDEX #2 (DEC 2) : DECELERATION RAMP
			EPL.FUB.EPLWrite_0.pData := ADR(EPL.Param.WriteData);  //POINTER TO THE DATA BEING WRITTEN
			EPL.FUB.EPLWrite_0.datalen := SIZEOF(EPL.Param.WriteData);  //SIZE OF THE DATA TO BE WRITTEN
			EPL.FUB.EPLWrite_0();

			IF EPL.FUB.EPLWrite_0.status = 0 THEN  //WRITE SUCCESSFUL
				EPL.FUB.EPLWrite_0.enable := 0;  //DISABLE THE FUB
				IF EPL.INV.DEC[1] THEN
					EPL.State := EPL_WAIT;
					EPL.INV.DECIndex := 0;
					InvPerms.CL1.Decel := InvTemps.CL1.Decel;
				ELSE
					EPL.State := EPL_INV2_ACCCHECK;
				END_IF
			ELSIF EPL.FUB.EPLWrite_0.status = ERR_FUB_BUSY THEN
				//BUSY
			ELSIF EPL.FUB.EPLWrite_0.status = ERR_FUB_ENABLE_FALSE THEN
				//DISABLED
			ELSE
				EPL.State := EPL_ERROR;
				EPL.INV.DECIndex := 0;
			END_IF

		EPL_INV2_ACCCHECK:
			IF(CS1.Module.OK) THEN
				IF(EPL.INV.ACC[2]) THEN
					IF(InvTemps.CS1.Accel <> InvPerms.CS1.Accel) THEN
						EPL.Param.WriteData := InvTemps.CS1.Accel;
						EPL.State := EPL_INV2_ACCWRITE;
					ELSE
						EPL.State := EPL_WAIT;
						EPL.INV.ACCIndex := 0;
					END_IF
				ELSE
					IF(InvPerms.CS1.Accel <> 5) THEN
						EPL.Param.WriteData := InvPerms.CS1.Accel;
						EPL.State := EPL_INV2_ACCWRITE;
					ELSE
						EPL.State := EPL_INV2_DECCHECK;
					END_IF
				END_IF
			END_IF

		EPL_INV2_ACCWRITE:

			EPL.FUB.EPLWrite_0.enable := 1;  //ENABLE FUB
			EPL.FUB.EPLWrite_0.pDevice := ADR('SL1.IF1.ST5');  //DEVICE NAME OF INVERTER
			EPL.FUB.EPLWrite_0.node := 5;  //NODE NUMBER OF THE STATION
			EPL.FUB.EPLWrite_0.index := 8252;  //WRITE INDEX 16#203C (DEC 8252)
			EPL.FUB.EPLWrite_0.subindex := 2;  //SUBINDEX #2 (DEC 2) : ACCELERATION RAMP
			EPL.FUB.EPLWrite_0.pData := ADR(EPL.Param.WriteData);  //POINTER TO THE DATA BEING WRITTEN
			EPL.FUB.EPLWrite_0.datalen := SIZEOF(EPL.Param.WriteData);  //SIZE OF THE DATA TO BE WRITTEN
			EPL.FUB.EPLWrite_0();

			IF EPL.FUB.EPLWrite_0.status = 0 THEN  //WRITE SUCCESSFUL
				EPL.FUB.EPLWrite_0.enable := 0;  //DISABLE THE FUB
				IF EPL.INV.ACC[2] THEN
					EPL.State := EPL_WAIT;
					EPL.INV.ACCIndex := 0;
					InvPerms.CS1.Accel := InvTemps.CS1.Accel;
				ELSE
					EPL.State := EPL_INV2_DECCHECK;
				END_IF
			ELSIF EPL.FUB.EPLWrite_0.status = ERR_FUB_BUSY THEN
				//BUSY
			ELSIF EPL.FUB.EPLWrite_0.status = ERR_FUB_ENABLE_FALSE THEN
				//DISABLED
			ELSE
				EPL.State := EPL_ERROR;
				EPL.INV.ACCIndex := 0;
			END_IF

		EPL_INV2_DECCHECK:
			IF(CS1.Module.OK) THEN
				IF(EPL.INV.DEC[2]) THEN
					IF(InvTemps.CS1.Decel <> InvPerms.CS1.Decel) THEN
						EPL.Param.WriteData := InvTemps.CS1.Decel;
						EPL.State := EPL_INV2_DECWRITE;
					ELSE
						EPL.State := EPL_WAIT;
						EPL.INV.DECIndex := 0;
					END_IF
				ELSE
					IF(InvPerms.CS1.Decel <> 5) THEN
						EPL.Param.WriteData := InvPerms.CS1.Decel;
						EPL.State := EPL_INV2_DECWRITE;
					ELSE
						EPL.State := EPL_INV3_ACCCHECK;
					END_IF
				END_IF
			END_IF

		EPL_INV2_DECWRITE:

			EPL.FUB.EPLWrite_0.enable := 1;  //ENABLE FUB
			EPL.FUB.EPLWrite_0.pDevice := ADR('SL1.IF1.ST5');  //DEVICE NAME OF INVERTER
			EPL.FUB.EPLWrite_0.node := 5;  //NODE NUMBER OF THE STATION
			EPL.FUB.EPLWrite_0.index := 8252;  //WRITE INDEX 16#203C (DEC 8252)
			EPL.FUB.EPLWrite_0.subindex := 3;  //SUBINDEX #2 (DEC 2) : DECELERATION RAMP
			EPL.FUB.EPLWrite_0.pData := ADR(EPL.Param.WriteData);  //POINTER TO THE DATA BEING WRITTEN
			EPL.FUB.EPLWrite_0.datalen := SIZEOF(EPL.Param.WriteData);  //SIZE OF THE DATA TO BE WRITTEN
			EPL.FUB.EPLWrite_0();

			IF EPL.FUB.EPLWrite_0.status = 0 THEN  //WRITE SUCCESSFUL
				EPL.FUB.EPLWrite_0.enable := 0;  //DISABLE THE FUB
				IF EPL.INV.DEC[2] THEN
					EPL.State := EPL_WAIT;
					EPL.INV.DECIndex := 0;
					InvPerms.CS1.Decel := InvTemps.CS1.Decel;
				ELSE
					EPL.State := EPL_INV3_ACCCHECK;
				END_IF
			ELSIF EPL.FUB.EPLWrite_0.status = ERR_FUB_BUSY THEN
				//BUSY
			ELSIF EPL.FUB.EPLWrite_0.status = ERR_FUB_ENABLE_FALSE THEN
				//DISABLED
			ELSE
				EPL.State := EPL_ERROR;
				EPL.INV.DECIndex := 0;
			END_IF

		EPL_INV3_ACCCHECK:
			IF(CV1.Module.OK) THEN
				IF(EPL.INV.ACC[3]) THEN
					IF(InvTemps.CV1.Accel <> InvPerms.CV1.Accel) THEN
						EPL.Param.WriteData := InvTemps.CV1.Accel;
						EPL.State := EPL_INV3_ACCWRITE;
					ELSE
						EPL.State := EPL_WAIT;
						EPL.INV.ACCIndex := 0;
					END_IF
				ELSE
					IF(InvPerms.CV1.Accel <> 5) THEN
						EPL.Param.WriteData := InvPerms.CV1.Accel;
						EPL.State := EPL_INV3_ACCWRITE;
					ELSE
						EPL.State := EPL_INV3_DECCHECK;
					END_IF
				END_IF
			END_IF

		EPL_INV3_ACCWRITE:

			EPL.FUB.EPLWrite_0.enable := 1;  //ENABLE FUB
			EPL.FUB.EPLWrite_0.pDevice := ADR('SL1.IF1.ST6');  //DEVICE NAME OF INVERTER
			EPL.FUB.EPLWrite_0.node := 6;  //NODE NUMBER OF THE STATION
			EPL.FUB.EPLWrite_0.index := 8252;  //WRITE INDEX 16#203C (DEC 8252)
			EPL.FUB.EPLWrite_0.subindex := 2;  //SUBINDEX #2 (DEC 2) : ACCELERATION RAMP
			EPL.FUB.EPLWrite_0.pData := ADR(EPL.Param.WriteData);  //POINTER TO THE DATA BEING WRITTEN
			EPL.FUB.EPLWrite_0.datalen := SIZEOF(EPL.Param.WriteData);  //SIZE OF THE DATA TO BE WRITTEN
			EPL.FUB.EPLWrite_0();

			IF EPL.FUB.EPLWrite_0.status = 0 THEN  //WRITE SUCCESSFUL
				EPL.FUB.EPLWrite_0.enable := 0;  //DISABLE THE FUB
				IF EPL.INV.ACC[3] THEN
					EPL.State := EPL_WAIT;
					EPL.INV.ACCIndex := 0;
					InvPerms.CV1.Accel := InvTemps.CV1.Accel;
				ELSE
					EPL.State := EPL_INV3_DECCHECK;
				END_IF
			ELSIF EPL.FUB.EPLWrite_0.status = ERR_FUB_BUSY THEN
				//BUSY
			ELSIF EPL.FUB.EPLWrite_0.status = ERR_FUB_ENABLE_FALSE THEN
				//DISABLED
			ELSE
				EPL.State := EPL_ERROR;
				EPL.INV.ACCIndex := 0;
			END_IF

		EPL_INV3_DECCHECK:
			IF(CV1.Module.OK) THEN
				IF(EPL.INV.DEC[3]) THEN
					IF(InvTemps.CV1.Decel <> InvPerms.CV1.Decel) THEN
						EPL.Param.WriteData := InvTemps.CV1.Decel;
						EPL.State := EPL_INV3_DECWRITE;
					ELSE
						EPL.State := EPL_WAIT;
						EPL.INV.DECIndex := 0;
					END_IF
				ELSE
					IF(InvPerms.CV1.Decel <> 5) THEN
						EPL.Param.WriteData := InvPerms.CV1.Decel;
						EPL.State := EPL_INV3_DECWRITE;
					ELSE
						EPL.State := EPL_INV4_ACCCHECK;
					END_IF
				END_IF
			END_IF

		EPL_INV3_DECWRITE:

			EPL.FUB.EPLWrite_0.enable := 1;  //ENABLE FUB
			EPL.FUB.EPLWrite_0.pDevice := ADR('SL1.IF1.ST6');  //DEVICE NAME OF INVERTER
			EPL.FUB.EPLWrite_0.node := 6;  //NODE NUMBER OF THE STATION
			EPL.FUB.EPLWrite_0.index := 8252;  //WRITE INDEX 16#203C (DEC 8252)
			EPL.FUB.EPLWrite_0.subindex := 3;  //SUBINDEX #2 (DEC 2) : DECELERATION RAMP
			EPL.FUB.EPLWrite_0.pData := ADR(EPL.Param.WriteData);  //POINTER TO THE DATA BEING WRITTEN
			EPL.FUB.EPLWrite_0.datalen := SIZEOF(EPL.Param.WriteData);  //SIZE OF THE DATA TO BE WRITTEN
			EPL.FUB.EPLWrite_0();

			IF EPL.FUB.EPLWrite_0.status = 0 THEN  //WRITE SUCCESSFUL
				EPL.FUB.EPLWrite_0.enable := 0;  //DISABLE THE FUB
				IF EPL.INV.DEC[3] THEN
					EPL.State := EPL_WAIT;
					EPL.INV.DECIndex := 0;
					InvPerms.CV1.Decel := InvTemps.CV1.Decel;
				ELSE
					EPL.State := EPL_INV4_ACCCHECK;
				END_IF
			ELSIF EPL.FUB.EPLWrite_0.status = ERR_FUB_BUSY THEN
				//BUSY
			ELSIF EPL.FUB.EPLWrite_0.status = ERR_FUB_ENABLE_FALSE THEN
				//DISABLED
			ELSE
				EPL.State := EPL_ERROR;
				EPL.INV.DECIndex := 0;
			END_IF

		EPL_INV4_ACCCHECK:
			IF(CC1.Module.OK) THEN
				IF(EPL.INV.ACC[4]) THEN
					IF(InvTemps.CC1.Accel <> InvPerms.CC1.Accel) THEN
						EPL.Param.WriteData := InvTemps.CC1.Accel;
						EPL.State := EPL_INV4_ACCWRITE;
					ELSE
						EPL.State := EPL_WAIT;
						EPL.INV.ACCIndex := 0;
					END_IF
				ELSE
					IF(InvPerms.CC1.Accel <> 5) THEN
						EPL.Param.WriteData := InvPerms.CC1.Accel;
						EPL.State := EPL_INV4_ACCWRITE;
					ELSE
						EPL.State := EPL_INV4_DECCHECK;
					END_IF
				END_IF
			END_IF

		EPL_INV4_ACCWRITE:

			EPL.FUB.EPLWrite_0.enable := 1;  //ENABLE FUB
			EPL.FUB.EPLWrite_0.pDevice := ADR('SL1.IF1.ST7');  //DEVICE NAME OF INVERTER
			EPL.FUB.EPLWrite_0.node := 7;  //NODE NUMBER OF THE STATION
			EPL.FUB.EPLWrite_0.index := 8252;  //WRITE INDEX 16#203C (DEC 8252)
			EPL.FUB.EPLWrite_0.subindex := 2;  //SUBINDEX #2 (DEC 2) : ACCELERATION RAMP
			EPL.FUB.EPLWrite_0.pData := ADR(EPL.Param.WriteData);  //POINTER TO THE DATA BEING WRITTEN
			EPL.FUB.EPLWrite_0.datalen := SIZEOF(EPL.Param.WriteData);  //SIZE OF THE DATA TO BE WRITTEN
			EPL.FUB.EPLWrite_0();

			IF EPL.FUB.EPLWrite_0.status = 0 THEN  //WRITE SUCCESSFUL
				EPL.FUB.EPLWrite_0.enable := 0;  //DISABLE THE FUB
				IF EPL.INV.ACC[4] THEN
					EPL.State := EPL_WAIT;
					EPL.INV.ACCIndex := 0;
					InvPerms.CC1.Accel := InvTemps.CC1.Accel;
				ELSE
					EPL.State := EPL_INV4_DECCHECK;
				END_IF
			ELSIF EPL.FUB.EPLWrite_0.status = ERR_FUB_BUSY THEN
				//BUSY
			ELSIF EPL.FUB.EPLWrite_0.status = ERR_FUB_ENABLE_FALSE THEN
				//DISABLED
			ELSE
				EPL.State := EPL_ERROR;
				EPL.INV.ACCIndex := 0;
			END_IF

		EPL_INV4_DECCHECK:
			IF(CC1.Module.OK) THEN
				IF(EPL.INV.DEC[4]) THEN
					IF(InvTemps.CC1.Decel <> InvPerms.CC1.Decel) THEN
						EPL.Param.WriteData := InvTemps.CC1.Decel;
						EPL.State := EPL_INV4_DECWRITE;
					ELSE
						EPL.State := EPL_WAIT;
						EPL.INV.DECIndex := 0;
					END_IF
				ELSE
					IF(InvPerms.CC1.Decel <> 5) THEN
						EPL.Param.WriteData := InvPerms.CC1.Decel;
						EPL.State := EPL_INV4_DECWRITE;
					ELSE
						EPL.State := EPL_INV5_ACCCHECK;
					END_IF
				END_IF
			END_IF

		EPL_INV4_DECWRITE:

			EPL.FUB.EPLWrite_0.enable := 1;  //ENABLE FUB
			EPL.FUB.EPLWrite_0.pDevice := ADR('SL1.IF1.ST7');  //DEVICE NAME OF INVERTER
			EPL.FUB.EPLWrite_0.node := 7;  //NODE NUMBER OF THE STATION
			EPL.FUB.EPLWrite_0.index := 8252;  //WRITE INDEX 16#203C (DEC 8252)
			EPL.FUB.EPLWrite_0.subindex := 3;  //SUBINDEX #2 (DEC 2) : DECELERATION RAMP
			EPL.FUB.EPLWrite_0.pData := ADR(EPL.Param.WriteData);  //POINTER TO THE DATA BEING WRITTEN
			EPL.FUB.EPLWrite_0.datalen := SIZEOF(EPL.Param.WriteData);  //SIZE OF THE DATA TO BE WRITTEN
			EPL.FUB.EPLWrite_0();

			IF EPL.FUB.EPLWrite_0.status = 0 THEN  //WRITE SUCCESSFUL
				EPL.FUB.EPLWrite_0.enable := 0;  //DISABLE THE FUB
				IF EPL.INV.DEC[4] THEN
					EPL.State := EPL_WAIT;
					EPL.INV.DECIndex := 0;
					InvPerms.CC1.Decel := InvTemps.CC1.Decel;
				ELSE
					EPL.State := EPL_INV5_ACCCHECK;
				END_IF
			ELSIF EPL.FUB.EPLWrite_0.status = ERR_FUB_BUSY THEN
				//BUSY
			ELSIF EPL.FUB.EPLWrite_0.status = ERR_FUB_ENABLE_FALSE THEN
				//DISABLED
			ELSE
				EPL.State := EPL_ERROR;
				EPL.INV.DECIndex := 0;
			END_IF

		EPL_INV5_ACCCHECK:
			IF(CC2.Module.OK) THEN
				IF(EPL.INV.ACC[5]) THEN
					IF(InvTemps.CC2.Accel <> InvPerms.CC2.Accel) THEN
						EPL.Param.WriteData := InvTemps.CC2.Accel;
						EPL.State := EPL_INV5_ACCWRITE;
					ELSE
						EPL.State := EPL_WAIT;
						EPL.INV.ACCIndex := 0;
					END_IF
				ELSE
					IF(InvPerms.CC2.Accel <> 5) THEN
						EPL.Param.WriteData := InvPerms.CC2.Accel;
						EPL.State := EPL_INV5_ACCWRITE;
					ELSE
						EPL.State := EPL_INV5_DECCHECK;
					END_IF
				END_IF
			END_IF

		EPL_INV5_ACCWRITE:

			EPL.FUB.EPLWrite_0.enable := 1;  //ENABLE FUB
			EPL.FUB.EPLWrite_0.pDevice := ADR('SL1.IF1.ST8');  //DEVICE NAME OF INVERTER
			EPL.FUB.EPLWrite_0.node := 8;  //NODE NUMBER OF THE STATION
			EPL.FUB.EPLWrite_0.index := 8252;  //WRITE INDEX 16#203C (DEC 8252)
			EPL.FUB.EPLWrite_0.subindex := 2;  //SUBINDEX #2 (DEC 2) : ACCELERATION RAMP
			EPL.FUB.EPLWrite_0.pData := ADR(EPL.Param.WriteData);  //POINTER TO THE DATA BEING WRITTEN
			EPL.FUB.EPLWrite_0.datalen := SIZEOF(EPL.Param.WriteData);  //SIZE OF THE DATA TO BE WRITTEN
			EPL.FUB.EPLWrite_0();

			IF EPL.FUB.EPLWrite_0.status = 0 THEN  //WRITE SUCCESSFUL
				EPL.FUB.EPLWrite_0.enable := 0;  //DISABLE THE FUB
				IF EPL.INV.ACC[5] THEN
					EPL.State := EPL_WAIT;
					EPL.INV.ACCIndex := 0;
					InvPerms.CC2.Accel := InvTemps.CC2.Accel;
				ELSE
					EPL.State := EPL_INV5_DECCHECK;
				END_IF
			ELSIF EPL.FUB.EPLWrite_0.status = ERR_FUB_BUSY THEN
				//BUSY
			ELSIF EPL.FUB.EPLWrite_0.status = ERR_FUB_ENABLE_FALSE THEN
				//DISABLED
			ELSE
				EPL.State := EPL_ERROR;
				EPL.INV.ACCIndex := 0;
			END_IF

		EPL_INV5_DECCHECK:
			IF(CC2.Module.OK) THEN
				IF(EPL.INV.DEC[5]) THEN
					IF(InvTemps.CC2.Decel <> InvPerms.CC2.Decel) THEN
						EPL.Param.WriteData := InvTemps.CC2.Decel;
						EPL.State := EPL_INV5_DECWRITE;
					ELSE
						EPL.State := EPL_WAIT;
						EPL.INV.DECIndex := 0;
					END_IF
				ELSE
					IF(InvPerms.CC2.Decel <> 5) THEN
						EPL.Param.WriteData := InvPerms.CC2.Decel;
						EPL.State := EPL_INV5_DECWRITE;
					ELSE
						EPL.State := EPL_INV6_ACCCHECK;
					END_IF
				END_IF
			END_IF

		EPL_INV5_DECWRITE:

			EPL.FUB.EPLWrite_0.enable := 1;  //ENABLE FUB
			EPL.FUB.EPLWrite_0.pDevice := ADR('SL1.IF1.ST8');  //DEVICE NAME OF INVERTER
			EPL.FUB.EPLWrite_0.node := 8;  //NODE NUMBER OF THE STATION
			EPL.FUB.EPLWrite_0.index := 8252;  //WRITE INDEX 16#203C (DEC 8252)
			EPL.FUB.EPLWrite_0.subindex := 3;  //SUBINDEX #2 (DEC 2) : DECELERATION RAMP
			EPL.FUB.EPLWrite_0.pData := ADR(EPL.Param.WriteData);  //POINTER TO THE DATA BEING WRITTEN
			EPL.FUB.EPLWrite_0.datalen := SIZEOF(EPL.Param.WriteData);  //SIZE OF THE DATA TO BE WRITTEN
			EPL.FUB.EPLWrite_0();

			IF EPL.FUB.EPLWrite_0.status = 0 THEN  //WRITE SUCCESSFUL
				EPL.FUB.EPLWrite_0.enable := 0;  //DISABLE THE FUB
				IF EPL.INV.DEC[5] THEN
					EPL.State := EPL_WAIT;
					EPL.INV.DECIndex := 0;
					InvPerms.CC2.Decel := InvTemps.CC2.Decel;
				ELSE
					EPL.State := EPL_INV6_ACCCHECK;
				END_IF
			ELSIF EPL.FUB.EPLWrite_0.status = ERR_FUB_BUSY THEN
				//BUSY
			ELSIF EPL.FUB.EPLWrite_0.status = ERR_FUB_ENABLE_FALSE THEN
				//DISABLED
			ELSE
				EPL.State := EPL_ERROR;
				EPL.INV.DECIndex := 0;
			END_IF

		EPL_INV6_ACCCHECK:
			IF(CS2.Module.OK) THEN
				IF(EPL.INV.ACC[6]) THEN
					IF(InvTemps.CS2.Accel <> InvPerms.CS2.Accel) THEN
						EPL.Param.WriteData := InvTemps.CS2.Accel;
						EPL.State := EPL_INV6_ACCWRITE;
					ELSE
						EPL.State := EPL_WAIT;
						EPL.INV.ACCIndex := 0;
					END_IF
				ELSE
					IF(InvPerms.CS2.Accel <> 5) THEN
						EPL.Param.WriteData := InvPerms.CS2.Accel;
						EPL.State := EPL_INV6_ACCWRITE;
					ELSE
						EPL.State := EPL_INV6_DECCHECK;
					END_IF
				END_IF
			END_IF

		EPL_INV6_ACCWRITE:

			EPL.FUB.EPLWrite_0.enable := 1;  //ENABLE FUB
			EPL.FUB.EPLWrite_0.pDevice := ADR('SL1.IF1.ST9');  //DEVICE NAME OF INVERTER
			EPL.FUB.EPLWrite_0.node := 9;  //NODE NUMBER OF THE STATION
			EPL.FUB.EPLWrite_0.index := 8252;  //WRITE INDEX 16#203C (DEC 8252)
			EPL.FUB.EPLWrite_0.subindex := 2;  //SUBINDEX #2 (DEC 2) : ACCELERATION RAMP
			EPL.FUB.EPLWrite_0.pData := ADR(EPL.Param.WriteData);  //POINTER TO THE DATA BEING WRITTEN
			EPL.FUB.EPLWrite_0.datalen := SIZEOF(EPL.Param.WriteData);  //SIZE OF THE DATA TO BE WRITTEN
			EPL.FUB.EPLWrite_0();

			IF EPL.FUB.EPLWrite_0.status = 0 THEN  //WRITE SUCCESSFUL
				EPL.FUB.EPLWrite_0.enable := 0;  //DISABLE THE FUB
				IF EPL.INV.ACC[6] THEN
					EPL.State := EPL_WAIT;
					EPL.INV.ACCIndex := 0;
					InvPerms.CS2.Accel := InvTemps.CS2.Accel;
				ELSE
					EPL.State := EPL_INV6_DECCHECK;
				END_IF
			ELSIF EPL.FUB.EPLWrite_0.status = ERR_FUB_BUSY THEN
				//BUSY
			ELSIF EPL.FUB.EPLWrite_0.status = ERR_FUB_ENABLE_FALSE THEN
				//DISABLED
			ELSE
				EPL.State := EPL_ERROR;
				EPL.INV.ACCIndex := 0;
			END_IF

		EPL_INV6_DECCHECK:
			IF(CS2.Module.OK) THEN
				IF(EPL.INV.DEC[6]) THEN
					IF(InvTemps.CS2.Decel <> InvPerms.CS2.Decel) THEN
						EPL.Param.WriteData := InvTemps.CS2.Decel;
						EPL.State := EPL_INV6_DECWRITE;
					ELSE
						EPL.State := EPL_WAIT;
						EPL.INV.DECIndex := 0;
					END_IF
				ELSE
					IF(InvPerms.CS2.Decel <> 5) THEN
						EPL.Param.WriteData := InvPerms.CS2.Decel;
						EPL.State := EPL_INV6_DECWRITE;
					ELSE
						EPL.State := EPL_INV7_ACCCHECK;
					END_IF
				END_IF
			END_IF

		EPL_INV6_DECWRITE:

			EPL.FUB.EPLWrite_0.enable := 1;  //ENABLE FUB
			EPL.FUB.EPLWrite_0.pDevice := ADR('SL1.IF1.ST9');  //DEVICE NAME OF INVERTER
			EPL.FUB.EPLWrite_0.node := 9;  //NODE NUMBER OF THE STATION
			EPL.FUB.EPLWrite_0.index := 8252;  //WRITE INDEX 16#203C (DEC 8252)
			EPL.FUB.EPLWrite_0.subindex := 3;  //SUBINDEX #2 (DEC 2) : DECELERATION RAMP
			EPL.FUB.EPLWrite_0.pData := ADR(EPL.Param.WriteData);  //POINTER TO THE DATA BEING WRITTEN
			EPL.FUB.EPLWrite_0.datalen := SIZEOF(EPL.Param.WriteData);  //SIZE OF THE DATA TO BE WRITTEN
			EPL.FUB.EPLWrite_0();

			IF EPL.FUB.EPLWrite_0.status = 0 THEN  //WRITE SUCCESSFUL
				EPL.FUB.EPLWrite_0.enable := 0;  //DISABLE THE FUB
				IF EPL.INV.DEC[6] THEN
					EPL.State := EPL_WAIT;
					EPL.INV.DECIndex := 0;
					InvPerms.CS2.Decel := InvTemps.CS2.Decel;
				ELSE
					EPL.State := EPL_INV7_ACCCHECK;
				END_IF
			ELSIF EPL.FUB.EPLWrite_0.status = ERR_FUB_BUSY THEN
				//BUSY
			ELSIF EPL.FUB.EPLWrite_0.status = ERR_FUB_ENABLE_FALSE THEN
				//DISABLED
			ELSE
				EPL.State := EPL_ERROR;
				EPL.INV.DECIndex := 0;
			END_IF

		EPL_INV7_ACCCHECK:
			IF(CV2.Module.OK) THEN
				IF(EPL.INV.ACC[7]) THEN
					IF(InvTemps.CV2.Accel <> InvPerms.CV2.Accel) THEN
						EPL.Param.WriteData := InvTemps.CV2.Accel;
						EPL.State := EPL_INV7_ACCWRITE;
					ELSE
						EPL.State := EPL_WAIT;
						EPL.INV.ACCIndex := 0;
					END_IF
				ELSE
					IF(InvPerms.CV2.Accel <> 5) THEN
						EPL.Param.WriteData := InvPerms.CV2.Accel;
						EPL.State := EPL_INV7_ACCWRITE;
					ELSE
						EPL.State := EPL_INV7_DECCHECK;
					END_IF
				END_IF
			END_IF

		EPL_INV7_ACCWRITE:

			EPL.FUB.EPLWrite_0.enable := 1;  //ENABLE FUB
			EPL.FUB.EPLWrite_0.pDevice := ADR('SL1.IF1.ST10');  //DEVICE NAME OF INVERTER
			EPL.FUB.EPLWrite_0.node := 10;  //NODE NUMBER OF THE STATION
			EPL.FUB.EPLWrite_0.index := 8252;  //WRITE INDEX 16#203C (DEC 8252)
			EPL.FUB.EPLWrite_0.subindex := 2;  //SUBINDEX #2 (DEC 2) : ACCELERATION RAMP
			EPL.FUB.EPLWrite_0.pData := ADR(EPL.Param.WriteData);  //POINTER TO THE DATA BEING WRITTEN
			EPL.FUB.EPLWrite_0.datalen := SIZEOF(EPL.Param.WriteData);  //SIZE OF THE DATA TO BE WRITTEN
			EPL.FUB.EPLWrite_0();

			IF EPL.FUB.EPLWrite_0.status = 0 THEN  //WRITE SUCCESSFUL
				EPL.FUB.EPLWrite_0.enable := 0;  //DISABLE THE FUB
				IF EPL.INV.ACC[7] THEN
					EPL.State := EPL_WAIT;
					EPL.INV.ACCIndex := 0;
					InvPerms.CV2.Accel := InvTemps.CV2.Accel;
				ELSE
					EPL.State := EPL_INV7_DECCHECK;
				END_IF
			ELSIF EPL.FUB.EPLWrite_0.status = ERR_FUB_BUSY THEN
				//BUSY
			ELSIF EPL.FUB.EPLWrite_0.status = ERR_FUB_ENABLE_FALSE THEN
				//DISABLED
			ELSE
				EPL.State := EPL_ERROR;
				EPL.INV.ACCIndex := 0;
			END_IF

		EPL_INV7_DECCHECK:
			IF(CV2.Module.OK) THEN
				IF(EPL.INV.DEC[7]) THEN
					IF(InvTemps.CV2.Decel <> InvPerms.CV2.Decel) THEN
						EPL.Param.WriteData := InvTemps.CV2.Decel;
						EPL.State := EPL_INV7_DECWRITE;
					ELSE
						EPL.State := EPL_WAIT;
						EPL.INV.DECIndex := 0;
					END_IF
				ELSE
					IF(InvPerms.CV2.Decel <> 5) THEN
						EPL.Param.WriteData := InvPerms.CV2.Decel;
						EPL.State := EPL_INV7_DECWRITE;
					ELSE
						EPL.State := EPL_INV8_ACCCHECK;
					END_IF
				END_IF
			END_IF

		EPL_INV7_DECWRITE:

			EPL.FUB.EPLWrite_0.enable := 1;  //ENABLE FUB
			EPL.FUB.EPLWrite_0.pDevice := ADR('SL1.IF1.ST10');  //DEVICE NAME OF INVERTER
			EPL.FUB.EPLWrite_0.node := 10;  //NODE NUMBER OF THE STATION
			EPL.FUB.EPLWrite_0.index := 8252;  //WRITE INDEX 16#203C (DEC 8252)
			EPL.FUB.EPLWrite_0.subindex := 3;  //SUBINDEX #2 (DEC 2) : DECELERATION RAMP
			EPL.FUB.EPLWrite_0.pData := ADR(EPL.Param.WriteData);  //POINTER TO THE DATA BEING WRITTEN
			EPL.FUB.EPLWrite_0.datalen := SIZEOF(EPL.Param.WriteData);  //SIZE OF THE DATA TO BE WRITTEN
			EPL.FUB.EPLWrite_0();

			IF EPL.FUB.EPLWrite_0.status = 0 THEN  //WRITE SUCCESSFUL
				EPL.FUB.EPLWrite_0.enable := 0;  //DISABLE THE FUB
				IF EPL.INV.DEC[7] THEN
					EPL.State := EPL_WAIT;
					EPL.INV.DECIndex := 0;
					InvPerms.CV2.Decel := InvTemps.CV2.Decel;
				ELSE
					EPL.State := EPL_INV8_ACCCHECK;
				END_IF
			ELSIF EPL.FUB.EPLWrite_0.status = ERR_FUB_BUSY THEN
				//BUSY
			ELSIF EPL.FUB.EPLWrite_0.status = ERR_FUB_ENABLE_FALSE THEN
				//DISABLED
			ELSE
				EPL.State := EPL_ERROR;
				EPL.INV.DECIndex := 0;
			END_IF

		EPL_INV8_ACCCHECK:
			IF(CC3.Module.OK) THEN
				IF(EPL.INV.ACC[8]) THEN
					IF(InvTemps.CC3.Accel <> InvPerms.CC3.Accel) THEN
						EPL.Param.WriteData := InvTemps.CC3.Accel;
						EPL.State := EPL_INV8_ACCWRITE;
					ELSE
						EPL.State := EPL_WAIT;
						EPL.INV.ACCIndex := 0;
					END_IF
				ELSE
					IF(InvPerms.CC3.Accel <> 5) THEN
						EPL.Param.WriteData := InvPerms.CC3.Accel;
						EPL.State := EPL_INV8_ACCWRITE;
					ELSE
						EPL.State := EPL_INV8_DECCHECK;
					END_IF
				END_IF
			END_IF

		EPL_INV8_ACCWRITE:

			EPL.FUB.EPLWrite_0.enable := 1;  //ENABLE FUB
			EPL.FUB.EPLWrite_0.pDevice := ADR('SL1.IF1.ST11');  //DEVICE NAME OF INVERTER
			EPL.FUB.EPLWrite_0.node := 11;  //NODE NUMBER OF THE STATION
			EPL.FUB.EPLWrite_0.index := 8252;  //WRITE INDEX 16#203C (DEC 8252)
			EPL.FUB.EPLWrite_0.subindex := 2;  //SUBINDEX #2 (DEC 2) : ACCELERATION RAMP
			EPL.FUB.EPLWrite_0.pData := ADR(EPL.Param.WriteData);  //POINTER TO THE DATA BEING WRITTEN
			EPL.FUB.EPLWrite_0.datalen := SIZEOF(EPL.Param.WriteData);  //SIZE OF THE DATA TO BE WRITTEN
			EPL.FUB.EPLWrite_0();

			IF EPL.FUB.EPLWrite_0.status = 0 THEN  //WRITE SUCCESSFUL
				EPL.FUB.EPLWrite_0.enable := 0;  //DISABLE THE FUB
				IF EPL.INV.ACC[8] THEN
					EPL.State := EPL_WAIT;
					EPL.INV.ACCIndex := 0;
					InvPerms.CC3.Accel := InvTemps.CC3.Accel;
				ELSE
					EPL.State := EPL_INV8_DECCHECK;
				END_IF
			ELSIF EPL.FUB.EPLWrite_0.status = ERR_FUB_BUSY THEN
				//BUSY
			ELSIF EPL.FUB.EPLWrite_0.status = ERR_FUB_ENABLE_FALSE THEN
				//DISABLED
			ELSE
				EPL.State := EPL_ERROR;
				EPL.INV.ACCIndex := 0;
			END_IF

		EPL_INV8_DECCHECK:
			IF(CC3.Module.OK) THEN
				IF(EPL.INV.DEC[8]) THEN
					IF(InvTemps.CC3.Decel <> InvPerms.CC3.Decel) THEN
						EPL.Param.WriteData := InvTemps.CC3.Decel;
						EPL.State := EPL_INV8_DECWRITE;
					ELSE
						EPL.State := EPL_WAIT;
						EPL.INV.DECIndex := 0;
					END_IF
				ELSE
					IF(InvPerms.CC3.Decel <> 5) THEN
						EPL.Param.WriteData := InvPerms.CC3.Decel;
						EPL.State := EPL_INV8_DECWRITE;
					ELSE
						EPL.State := EPL_INV9_ACCCHECK;
					END_IF
				END_IF
			END_IF

		EPL_INV8_DECWRITE:

			EPL.FUB.EPLWrite_0.enable := 1;  //ENABLE FUB
			EPL.FUB.EPLWrite_0.pDevice := ADR('SL1.IF1.ST11');  //DEVICE NAME OF INVERTER
			EPL.FUB.EPLWrite_0.node := 11;  //NODE NUMBER OF THE STATION
			EPL.FUB.EPLWrite_0.index := 8252;  //WRITE INDEX 16#203C (DEC 8252)
			EPL.FUB.EPLWrite_0.subindex := 3;  //SUBINDEX #2 (DEC 2) : DECELERATION RAMP
			EPL.FUB.EPLWrite_0.pData := ADR(EPL.Param.WriteData);  //POINTER TO THE DATA BEING WRITTEN
			EPL.FUB.EPLWrite_0.datalen := SIZEOF(EPL.Param.WriteData);  //SIZE OF THE DATA TO BE WRITTEN
			EPL.FUB.EPLWrite_0();

			IF EPL.FUB.EPLWrite_0.status = 0 THEN  //WRITE SUCCESSFUL
				EPL.FUB.EPLWrite_0.enable := 0;  //DISABLE THE FUB
				IF EPL.INV.DEC[8] THEN
					EPL.State := EPL_WAIT;
					EPL.INV.DECIndex := 0;
					InvPerms.CC3.Decel := InvTemps.CC3.Decel;
				ELSE
					EPL.State := EPL_INV9_ACCCHECK;
				END_IF
			ELSIF EPL.FUB.EPLWrite_0.status = ERR_FUB_BUSY THEN
				//BUSY
			ELSIF EPL.FUB.EPLWrite_0.status = ERR_FUB_ENABLE_FALSE THEN
				//DISABLED
			ELSE
				EPL.State := EPL_ERROR;
				EPL.INV.DECIndex := 0;
			END_IF

		EPL_INV9_ACCCHECK:
			IF(CC4.Module.OK) THEN
				IF(EPL.INV.ACC[9]) THEN
					IF(InvTemps.CC4.Accel <> InvPerms.CC4.Accel) THEN
						EPL.Param.WriteData := InvTemps.CC4.Accel;
						EPL.State := EPL_INV9_ACCWRITE;
					ELSE
						EPL.State := EPL_WAIT;
						EPL.INV.ACCIndex := 0;
					END_IF
				ELSE
					IF(InvPerms.CC4.Accel <> 5) THEN
						EPL.Param.WriteData := InvPerms.CC4.Accel;
						EPL.State := EPL_INV9_ACCWRITE;
					ELSE
						EPL.State := EPL_INV9_DECCHECK;
					END_IF
				END_IF
			END_IF

		EPL_INV9_ACCWRITE:

			EPL.FUB.EPLWrite_0.enable := 1;  //ENABLE FUB
			EPL.FUB.EPLWrite_0.pDevice := ADR('SL1.IF1.ST12');  //DEVICE NAME OF INVERTER
			EPL.FUB.EPLWrite_0.node := 12;  //NODE NUMBER OF THE STATION
			EPL.FUB.EPLWrite_0.index := 8252;  //WRITE INDEX 16#203C (DEC 8252)
			EPL.FUB.EPLWrite_0.subindex := 2;  //SUBINDEX #2 (DEC 2) : ACCELERATION RAMP
			EPL.FUB.EPLWrite_0.pData := ADR(EPL.Param.WriteData);  //POINTER TO THE DATA BEING WRITTEN
			EPL.FUB.EPLWrite_0.datalen := SIZEOF(EPL.Param.WriteData);  //SIZE OF THE DATA TO BE WRITTEN
			EPL.FUB.EPLWrite_0();

			IF EPL.FUB.EPLWrite_0.status = 0 THEN  //WRITE SUCCESSFUL
				EPL.FUB.EPLWrite_0.enable := 0;  //DISABLE THE FUB
				IF EPL.INV.ACC[9] THEN
					EPL.State := EPL_WAIT;
					EPL.INV.ACCIndex := 0;
					InvPerms.CC4.Accel := InvTemps.CC4.Accel;
				ELSE
					EPL.State := EPL_INV9_DECCHECK;
				END_IF
			ELSIF EPL.FUB.EPLWrite_0.status = ERR_FUB_BUSY THEN
				//BUSY
			ELSIF EPL.FUB.EPLWrite_0.status = ERR_FUB_ENABLE_FALSE THEN
				//DISABLED
			ELSE
				EPL.State := EPL_ERROR;
				EPL.INV.ACCIndex := 0;
			END_IF

		EPL_INV9_DECCHECK:
			IF(CC4.Module.OK) THEN
				IF(EPL.INV.DEC[9]) THEN
					IF(InvTemps.CC4.Decel <> InvPerms.CC4.Decel) THEN
						EPL.Param.WriteData := InvTemps.CC4.Decel;
						EPL.State := EPL_INV9_DECWRITE;
					ELSE
						EPL.State := EPL_WAIT;
						EPL.INV.DECIndex := 0;
					END_IF
				ELSE
					IF(InvPerms.CC4.Decel <> 5) THEN
						EPL.Param.WriteData := InvPerms.CC4.Decel;
						EPL.State := EPL_INV9_DECWRITE;
					ELSE
						EPL.State := EPL_INV10_ACCCHECK;
					END_IF
				END_IF
			END_IF

		EPL_INV9_DECWRITE:

			EPL.FUB.EPLWrite_0.enable := 1;  //ENABLE FUB
			EPL.FUB.EPLWrite_0.pDevice := ADR('SL1.IF1.ST12');  //DEVICE NAME OF INVERTER
			EPL.FUB.EPLWrite_0.node := 12;  //NODE NUMBER OF THE STATION
			EPL.FUB.EPLWrite_0.index := 8252;  //WRITE INDEX 16#203C (DEC 8252)
			EPL.FUB.EPLWrite_0.subindex := 3;  //SUBINDEX #2 (DEC 2) : DECELERATION RAMP
			EPL.FUB.EPLWrite_0.pData := ADR(EPL.Param.WriteData);  //POINTER TO THE DATA BEING WRITTEN
			EPL.FUB.EPLWrite_0.datalen := SIZEOF(EPL.Param.WriteData);  //SIZE OF THE DATA TO BE WRITTEN
			EPL.FUB.EPLWrite_0();

			IF EPL.FUB.EPLWrite_0.status = 0 THEN  //WRITE SUCCESSFUL
				EPL.FUB.EPLWrite_0.enable := 0;  //DISABLE THE FUB
				IF EPL.INV.DEC[9] THEN
					EPL.State := EPL_WAIT;
					EPL.INV.DECIndex := 0;
					InvPerms.CC4.Decel := InvTemps.CC4.Decel;
				ELSE
					EPL.State := EPL_INV10_ACCCHECK;
				END_IF
			ELSIF EPL.FUB.EPLWrite_0.status = ERR_FUB_BUSY THEN
				//BUSY
			ELSIF EPL.FUB.EPLWrite_0.status = ERR_FUB_ENABLE_FALSE THEN
				//DISABLED
			ELSE
				EPL.State := EPL_ERROR;
				EPL.INV.DECIndex := 0;
			END_IF

		EPL_INV10_ACCCHECK:
			IF(CB1.Module.OK) THEN
				IF(EPL.INV.ACC[10]) THEN
					IF(InvTemps.CB1.Accel <> InvPerms.CB1.Accel) THEN
						EPL.Param.WriteData := InvTemps.CB1.Accel;
						EPL.State := EPL_INV10_ACCWRITE;
					ELSE
						EPL.State := EPL_WAIT;
						EPL.INV.ACCIndex := 0;
					END_IF
				ELSE
					IF(InvPerms.CB1.Accel <> 5) THEN
						EPL.Param.WriteData := InvPerms.CB1.Accel;
						EPL.State := EPL_INV10_ACCWRITE;
					ELSE
						EPL.State := EPL_INV10_DECCHECK;
					END_IF
				END_IF
			END_IF

		EPL_INV10_ACCWRITE:

			EPL.FUB.EPLWrite_0.enable := 1;  //ENABLE FUB
			EPL.FUB.EPLWrite_0.pDevice := ADR('SL1.IF1.ST13');  //DEVICE NAME OF INVERTER
			EPL.FUB.EPLWrite_0.node := 13;  //NODE NUMBER OF THE STATION
			EPL.FUB.EPLWrite_0.index := 8252;  //WRITE INDEX 16#203C (DEC 8252)
			EPL.FUB.EPLWrite_0.subindex := 2;  //SUBINDEX #2 (DEC 2) : ACCELERATION RAMP
			EPL.FUB.EPLWrite_0.pData := ADR(EPL.Param.WriteData);  //POINTER TO THE DATA BEING WRITTEN
			EPL.FUB.EPLWrite_0.datalen := SIZEOF(EPL.Param.WriteData);  //SIZE OF THE DATA TO BE WRITTEN
			EPL.FUB.EPLWrite_0();

			IF EPL.FUB.EPLWrite_0.status = 0 THEN  //WRITE SUCCESSFUL
				EPL.FUB.EPLWrite_0.enable := 0;  //DISABLE THE FUB
				IF EPL.INV.ACC[10] THEN
					EPL.State := EPL_WAIT;
					EPL.INV.ACCIndex := 0;
					InvPerms.CB1.Accel := InvTemps.CB1.Accel;
				ELSE
					EPL.State := EPL_INV10_DECCHECK;
				END_IF
			ELSIF EPL.FUB.EPLWrite_0.status = ERR_FUB_BUSY THEN
				//BUSY
			ELSIF EPL.FUB.EPLWrite_0.status = ERR_FUB_ENABLE_FALSE THEN
				//DISABLED
			ELSE
				EPL.State := EPL_ERROR;
				EPL.INV.ACCIndex := 0;
			END_IF

		EPL_INV10_DECCHECK:
			IF(CB1.Module.OK) THEN
				IF(EPL.INV.DEC[10]) THEN
					IF(InvTemps.CB1.Decel <> InvPerms.CB1.Decel) THEN
						EPL.Param.WriteData := InvTemps.CB1.Decel;
						EPL.State := EPL_INV10_DECWRITE;
					ELSE
						EPL.State := EPL_WAIT;
						EPL.INV.DECIndex := 0;
					END_IF
				ELSE
					IF(InvPerms.CB1.Decel <> 5) THEN
						EPL.Param.WriteData := InvPerms.CB1.Decel;
						EPL.State := EPL_INV10_DECWRITE;
					ELSE
						EPL.State := EPL_INV11_ACCCHECK;
					END_IF
				END_IF
			END_IF

		EPL_INV10_DECWRITE:

			EPL.FUB.EPLWrite_0.enable := 1;  //ENABLE FUB
			EPL.FUB.EPLWrite_0.pDevice := ADR('SL1.IF1.ST13');  //DEVICE NAME OF INVERTER
			EPL.FUB.EPLWrite_0.node := 13;  //NODE NUMBER OF THE STATION
			EPL.FUB.EPLWrite_0.index := 8252;  //WRITE INDEX 16#203C (DEC 8252)
			EPL.FUB.EPLWrite_0.subindex := 3;  //SUBINDEX #2 (DEC 2) : DECELERATION RAMP
			EPL.FUB.EPLWrite_0.pData := ADR(EPL.Param.WriteData);  //POINTER TO THE DATA BEING WRITTEN
			EPL.FUB.EPLWrite_0.datalen := SIZEOF(EPL.Param.WriteData);  //SIZE OF THE DATA TO BE WRITTEN
			EPL.FUB.EPLWrite_0();

			IF EPL.FUB.EPLWrite_0.status = 0 THEN  //WRITE SUCCESSFUL
				EPL.FUB.EPLWrite_0.enable := 0;  //DISABLE THE FUB
				IF EPL.INV.DEC[10] THEN
					EPL.State := EPL_WAIT;
					EPL.INV.DECIndex := 0;
					InvPerms.CB1.Decel := InvTemps.CB1.Decel;
				ELSE
					EPL.State := EPL_INV11_ACCCHECK;
				END_IF
			ELSIF EPL.FUB.EPLWrite_0.status = ERR_FUB_BUSY THEN
				//BUSY
			ELSIF EPL.FUB.EPLWrite_0.status = ERR_FUB_ENABLE_FALSE THEN
				//DISABLED
			ELSE
				EPL.State := EPL_ERROR;
				EPL.INV.DECIndex := 0;
			END_IF

		EPL_INV11_ACCCHECK:
			IF(CB2.Module.OK) THEN
				IF(EPL.INV.ACC[11]) THEN
					IF(InvTemps.CB2.Accel <> InvPerms.CB2.Accel) THEN
						EPL.Param.WriteData := InvTemps.CB2.Accel;
						EPL.State := EPL_INV11_ACCWRITE;
					ELSE
						EPL.State := EPL_WAIT;
						EPL.INV.ACCIndex := 0;
					END_IF
				ELSE
					IF(InvPerms.CB2.Accel <> 5) THEN
						EPL.Param.WriteData := InvPerms.CB2.Accel;
						EPL.State := EPL_INV11_ACCWRITE;
					ELSE
						EPL.State := EPL_INV11_DECCHECK;
					END_IF
				END_IF
			END_IF

		EPL_INV11_ACCWRITE:

			EPL.FUB.EPLWrite_0.enable := 1;  //ENABLE FUB
			EPL.FUB.EPLWrite_0.pDevice := ADR('SL1.IF1.ST14');  //DEVICE NAME OF INVERTER
			EPL.FUB.EPLWrite_0.node := 14;  //NODE NUMBER OF THE STATION
			EPL.FUB.EPLWrite_0.index := 8252;  //WRITE INDEX 16#203C (DEC 8252)
			EPL.FUB.EPLWrite_0.subindex := 2;  //SUBINDEX #2 (DEC 2) : ACCELERATION RAMP
			EPL.FUB.EPLWrite_0.pData := ADR(EPL.Param.WriteData);  //POINTER TO THE DATA BEING WRITTEN
			EPL.FUB.EPLWrite_0.datalen := SIZEOF(EPL.Param.WriteData);  //SIZE OF THE DATA TO BE WRITTEN
			EPL.FUB.EPLWrite_0();

			IF EPL.FUB.EPLWrite_0.status = 0 THEN  //WRITE SUCCESSFUL
				EPL.FUB.EPLWrite_0.enable := 0;  //DISABLE THE FUB
				IF EPL.INV.ACC[11] THEN
					EPL.State := EPL_WAIT;
					EPL.INV.ACCIndex := 0;
					InvPerms.CB2.Accel := InvTemps.CB2.Accel;
				ELSE
					EPL.State := EPL_INV11_DECCHECK;
				END_IF
			ELSIF EPL.FUB.EPLWrite_0.status = ERR_FUB_BUSY THEN
				//BUSY
			ELSIF EPL.FUB.EPLWrite_0.status = ERR_FUB_ENABLE_FALSE THEN
				//DISABLED
			ELSE
				EPL.State := EPL_ERROR;
				EPL.INV.ACCIndex := 0;
			END_IF

		EPL_INV11_DECCHECK:
			IF(CB2.Module.OK) THEN
				IF(EPL.INV.DEC[11]) THEN
					IF(InvTemps.CB2.Decel <> InvPerms.CB2.Decel) THEN
						EPL.Param.WriteData := InvTemps.CB2.Decel;
						EPL.State := EPL_INV11_DECWRITE;
					ELSE
						EPL.State := EPL_WAIT;
						EPL.INV.DECIndex := 0;
					END_IF
				ELSE
					IF(InvPerms.CB2.Decel <> 5) THEN
						EPL.Param.WriteData := InvPerms.CB2.Decel;
						EPL.State := EPL_INV11_DECWRITE;
					ELSE
						EPL.State := EPL_INV12_ACCCHECK;
					END_IF
				END_IF
			END_IF

		EPL_INV11_DECWRITE:

			EPL.FUB.EPLWrite_0.enable := 1;  //ENABLE FUB
			EPL.FUB.EPLWrite_0.pDevice := ADR('SL1.IF1.ST14');  //DEVICE NAME OF INVERTER
			EPL.FUB.EPLWrite_0.node := 14;  //NODE NUMBER OF THE STATION
			EPL.FUB.EPLWrite_0.index := 8252;  //WRITE INDEX 16#203C (DEC 8252)
			EPL.FUB.EPLWrite_0.subindex := 3;  //SUBINDEX #2 (DEC 2) : DECELERATION RAMP
			EPL.FUB.EPLWrite_0.pData := ADR(EPL.Param.WriteData);  //POINTER TO THE DATA BEING WRITTEN
			EPL.FUB.EPLWrite_0.datalen := SIZEOF(EPL.Param.WriteData);  //SIZE OF THE DATA TO BE WRITTEN
			EPL.FUB.EPLWrite_0();

			IF EPL.FUB.EPLWrite_0.status = 0 THEN  //WRITE SUCCESSFUL
				EPL.FUB.EPLWrite_0.enable := 0;  //DISABLE THE FUB
				IF EPL.INV.DEC[11] THEN
					EPL.State := EPL_WAIT;
					EPL.INV.DECIndex := 0;
					InvPerms.CB2.Decel := InvTemps.CB2.Decel;
				ELSE
					EPL.State := EPL_INV12_ACCCHECK;
				END_IF
			ELSIF EPL.FUB.EPLWrite_0.status = ERR_FUB_BUSY THEN
				//BUSY
			ELSIF EPL.FUB.EPLWrite_0.status = ERR_FUB_ENABLE_FALSE THEN
				//DISABLED
			ELSE
				EPL.State := EPL_ERROR;
				EPL.INV.DECIndex := 0;
			END_IF

		EPL_INV12_ACCCHECK:
			IF(CRB.Module.OK) THEN
				IF(EPL.INV.ACC[12]) THEN
					IF(InvTemps.CRB.Accel <> InvPerms.CRB.Accel) THEN
						EPL.Param.WriteData := InvTemps.CRB.Accel;
						EPL.State := EPL_INV12_ACCWRITE;
					ELSE
						EPL.State := EPL_WAIT;
						EPL.INV.ACCIndex := 0;
					END_IF
				ELSE
					IF(InvPerms.CRB.Accel <> 5) THEN
						EPL.Param.WriteData := InvPerms.CRB.Accel;
						EPL.State := EPL_INV12_ACCWRITE;
					ELSE
						EPL.State := EPL_INV12_DECCHECK;
					END_IF
				END_IF
			END_IF

		EPL_INV12_ACCWRITE:

			EPL.FUB.EPLWrite_0.enable := 1;  //ENABLE FUB
			EPL.FUB.EPLWrite_0.pDevice := ADR('SL1.IF1.ST15');  //DEVICE NAME OF INVERTER
			EPL.FUB.EPLWrite_0.node := 15;  //NODE NUMBER OF THE STATION
			EPL.FUB.EPLWrite_0.index := 8252;  //WRITE INDEX 16#203C (DEC 8252)
			EPL.FUB.EPLWrite_0.subindex := 2;  //SUBINDEX #2 (DEC 2) : ACCELERATION RAMP
			EPL.FUB.EPLWrite_0.pData := ADR(EPL.Param.WriteData);  //POINTER TO THE DATA BEING WRITTEN
			EPL.FUB.EPLWrite_0.datalen := SIZEOF(EPL.Param.WriteData);  //SIZE OF THE DATA TO BE WRITTEN
			EPL.FUB.EPLWrite_0();

			IF EPL.FUB.EPLWrite_0.status = 0 THEN  //WRITE SUCCESSFUL
				EPL.FUB.EPLWrite_0.enable := 0;  //DISABLE THE FUB
				IF EPL.INV.ACC[12] THEN
					EPL.State := EPL_WAIT;
					EPL.INV.ACCIndex := 0;
					InvPerms.CRB.Accel := InvTemps.CRB.Accel;
				ELSE
					EPL.State := EPL_INV12_DECCHECK;
				END_IF
			ELSIF EPL.FUB.EPLWrite_0.status = ERR_FUB_BUSY THEN
				//BUSY
			ELSIF EPL.FUB.EPLWrite_0.status = ERR_FUB_ENABLE_FALSE THEN
				//DISABLED
			ELSE
				EPL.State := EPL_ERROR;
				EPL.INV.ACCIndex := 0;
			END_IF

		EPL_INV12_DECCHECK:
			IF(CRB.Module.OK) THEN
				IF(EPL.INV.DEC[12]) THEN
					IF(InvTemps.CRB.Decel <> InvPerms.CRB.Decel) THEN
						EPL.Param.WriteData := InvTemps.CRB.Decel;
						EPL.State := EPL_INV12_DECWRITE;
					ELSE
						EPL.State := EPL_WAIT;
						EPL.INV.DECIndex := 0;
					END_IF
				ELSE
					IF(InvPerms.CRB.Decel <> 5) THEN
						EPL.Param.WriteData := InvPerms.CRB.Decel;
						EPL.State := EPL_INV12_DECWRITE;
					ELSE
						EPL.State := EPL_INV13_ACCCHECK;
					END_IF
				END_IF
			END_IF

		EPL_INV12_DECWRITE:

			EPL.FUB.EPLWrite_0.enable := 1;  //ENABLE FUB
			EPL.FUB.EPLWrite_0.pDevice := ADR('SL1.IF1.ST15');  //DEVICE NAME OF INVERTER
			EPL.FUB.EPLWrite_0.node := 15;  //NODE NUMBER OF THE STATION
			EPL.FUB.EPLWrite_0.index := 8252;  //WRITE INDEX 16#203C (DEC 8252)
			EPL.FUB.EPLWrite_0.subindex := 3;  //SUBINDEX #2 (DEC 2) : DECELERATION RAMP
			EPL.FUB.EPLWrite_0.pData := ADR(EPL.Param.WriteData);  //POINTER TO THE DATA BEING WRITTEN
			EPL.FUB.EPLWrite_0.datalen := SIZEOF(EPL.Param.WriteData);  //SIZE OF THE DATA TO BE WRITTEN
			EPL.FUB.EPLWrite_0();

			IF EPL.FUB.EPLWrite_0.status = 0 THEN  //WRITE SUCCESSFUL
				EPL.FUB.EPLWrite_0.enable := 0;  //DISABLE THE FUB
				IF EPL.INV.DEC[12] THEN
					EPL.State := EPL_WAIT;
					EPL.INV.DECIndex := 0;
					InvPerms.CRB.Decel := InvTemps.CRB.Decel;
				ELSE
					EPL.State := EPL_INV13_ACCCHECK;
				END_IF
			ELSIF EPL.FUB.EPLWrite_0.status = ERR_FUB_BUSY THEN
				//BUSY
			ELSIF EPL.FUB.EPLWrite_0.status = ERR_FUB_ENABLE_FALSE THEN
				//DISABLED
			ELSE
				EPL.State := EPL_ERROR;
				EPL.INV.DECIndex := 0;
			END_IF

		EPL_INV13_ACCCHECK:
			IF(CRE.Module.OK) THEN
				IF(EPL.INV.ACC[13]) THEN
					IF(InvTemps.CRE.Accel <> InvPerms.CRE.Accel) THEN
						EPL.Param.WriteData := InvTemps.CRE.Accel;
						EPL.State := EPL_INV13_ACCWRITE;
					ELSE
						EPL.State := EPL_WAIT;
						EPL.INV.ACCIndex := 0;
					END_IF
				ELSE
					IF(InvPerms.CRE.Accel <> 5) THEN
						EPL.Param.WriteData := InvPerms.CRE.Accel;
						EPL.State := EPL_INV13_ACCWRITE;
					ELSE
						EPL.State := EPL_INV13_DECCHECK;
					END_IF
				END_IF
			END_IF

		EPL_INV13_ACCWRITE:

			EPL.FUB.EPLWrite_0.enable := 1;  //ENABLE FUB
			EPL.FUB.EPLWrite_0.pDevice := ADR('SL1.IF1.ST16');  //DEVICE NAME OF INVERTER
			EPL.FUB.EPLWrite_0.node := 16;  //NODE NUMBER OF THE STATION
			EPL.FUB.EPLWrite_0.index := 8252;  //WRITE INDEX 16#203C (DEC 8252)
			EPL.FUB.EPLWrite_0.subindex := 2;  //SUBINDEX #2 (DEC 2) : ACCELERATION RAMP
			EPL.FUB.EPLWrite_0.pData := ADR(EPL.Param.WriteData);  //POINTER TO THE DATA BEING WRITTEN
			EPL.FUB.EPLWrite_0.datalen := SIZEOF(EPL.Param.WriteData);  //SIZE OF THE DATA TO BE WRITTEN
			EPL.FUB.EPLWrite_0();

			IF EPL.FUB.EPLWrite_0.status = 0 THEN  //WRITE SUCCESSFUL
				EPL.FUB.EPLWrite_0.enable := 0;  //DISABLE THE FUB
				IF EPL.INV.ACC[13] THEN
					EPL.State := EPL_WAIT;
					EPL.INV.ACCIndex := 0;
					InvPerms.CRE.Accel := InvTemps.CRE.Accel;
				ELSE
					EPL.State := EPL_INV13_DECCHECK;
				END_IF
			ELSIF EPL.FUB.EPLWrite_0.status = ERR_FUB_BUSY THEN
				//BUSY
			ELSIF EPL.FUB.EPLWrite_0.status = ERR_FUB_ENABLE_FALSE THEN
				//DISABLED
			ELSE
				EPL.State := EPL_ERROR;
				EPL.INV.ACCIndex := 0;
			END_IF

		EPL_INV13_DECCHECK:
			IF(CRE.Module.OK) THEN
				IF(EPL.INV.DEC[13]) THEN
					IF(InvTemps.CRE.Decel <> InvPerms.CRE.Decel) THEN
						EPL.Param.WriteData := InvTemps.CRE.Decel;
						EPL.State := EPL_INV13_DECWRITE;
					ELSE
						EPL.State := EPL_WAIT;
						EPL.INV.DECIndex := 0;
					END_IF
				ELSE
					IF(InvPerms.CRE.Decel <> 5) THEN
						EPL.Param.WriteData := InvPerms.CRE.Decel;
						EPL.State := EPL_INV13_DECWRITE;
					ELSE
						EPL.State := EPL_INV14_ACCCHECK;
					END_IF
				END_IF
			END_IF

		EPL_INV13_DECWRITE:

			EPL.FUB.EPLWrite_0.enable := 1;  //ENABLE FUB
			EPL.FUB.EPLWrite_0.pDevice := ADR('SL1.IF1.ST16');  //DEVICE NAME OF INVERTER
			EPL.FUB.EPLWrite_0.node := 16;  //NODE NUMBER OF THE STATION
			EPL.FUB.EPLWrite_0.index := 8252;  //WRITE INDEX 16#203C (DEC 8252)
			EPL.FUB.EPLWrite_0.subindex := 3;  //SUBINDEX #2 (DEC 2) : DECELERATION RAMP
			EPL.FUB.EPLWrite_0.pData := ADR(EPL.Param.WriteData);  //POINTER TO THE DATA BEING WRITTEN
			EPL.FUB.EPLWrite_0.datalen := SIZEOF(EPL.Param.WriteData);  //SIZE OF THE DATA TO BE WRITTEN
			EPL.FUB.EPLWrite_0();

			IF EPL.FUB.EPLWrite_0.status = 0 THEN  //WRITE SUCCESSFUL
				EPL.FUB.EPLWrite_0.enable := 0;  //DISABLE THE FUB
				IF EPL.INV.DEC[13] THEN
					EPL.State := EPL_WAIT;
					EPL.INV.DECIndex := 0;
					InvPerms.CRE.Decel := InvTemps.CRE.Decel;
				ELSE
					EPL.State := EPL_INV14_ACCCHECK;
				END_IF
			ELSIF EPL.FUB.EPLWrite_0.status = ERR_FUB_BUSY THEN
				//BUSY
			ELSIF EPL.FUB.EPLWrite_0.status = ERR_FUB_ENABLE_FALSE THEN
				//DISABLED
			ELSE
				EPL.State := EPL_ERROR;
				EPL.INV.DECIndex := 0;
			END_IF

		EPL_INV14_ACCCHECK:
			IF(CLB.Module.OK) THEN
				IF(EPL.INV.ACC[14]) THEN
					IF(InvTemps.CLB.Accel <> InvPerms.CLB.Accel) THEN
						EPL.Param.WriteData := InvTemps.CLB.Accel;
						EPL.State := EPL_INV14_ACCWRITE;
					ELSE
						EPL.State := EPL_WAIT;
						EPL.INV.ACCIndex := 0;
					END_IF
				ELSE
					IF(InvPerms.CLB.Accel <> 5) THEN
						EPL.Param.WriteData := InvPerms.CLB.Accel;
						EPL.State := EPL_INV14_ACCWRITE;
					ELSE
						EPL.State := EPL_INV14_DECCHECK;
					END_IF
				END_IF
			END_IF

		EPL_INV14_ACCWRITE:

			EPL.FUB.EPLWrite_0.enable := 1;  //ENABLE FUB
			EPL.FUB.EPLWrite_0.pDevice := ADR('SL1.IF1.ST17');  //DEVICE NAME OF INVERTER
			EPL.FUB.EPLWrite_0.node := 17;  //NODE NUMBER OF THE STATION
			EPL.FUB.EPLWrite_0.index := 8252;  //WRITE INDEX 16#203C (DEC 8252)
			EPL.FUB.EPLWrite_0.subindex := 2;  //SUBINDEX #2 (DEC 2) : ACCELERATION RAMP
			EPL.FUB.EPLWrite_0.pData := ADR(EPL.Param.WriteData);  //POINTER TO THE DATA BEING WRITTEN
			EPL.FUB.EPLWrite_0.datalen := SIZEOF(EPL.Param.WriteData);  //SIZE OF THE DATA TO BE WRITTEN
			EPL.FUB.EPLWrite_0();

			IF EPL.FUB.EPLWrite_0.status = 0 THEN  //WRITE SUCCESSFUL
				EPL.FUB.EPLWrite_0.enable := 0;  //DISABLE THE FUB
				IF EPL.INV.ACC[14] THEN
					EPL.State := EPL_WAIT;
					EPL.INV.ACCIndex := 0;
					InvPerms.CLB.Accel := InvTemps.CLB.Accel;
				ELSE
					EPL.State := EPL_INV14_DECCHECK;
				END_IF
			ELSIF EPL.FUB.EPLWrite_0.status = ERR_FUB_BUSY THEN
				//BUSY
			ELSIF EPL.FUB.EPLWrite_0.status = ERR_FUB_ENABLE_FALSE THEN
				//DISABLED
			ELSE
				EPL.State := EPL_ERROR;
				EPL.INV.ACCIndex := 0;
			END_IF

		EPL_INV14_DECCHECK:
			IF(CLB.Module.OK) THEN
				IF(EPL.INV.DEC[14]) THEN
					IF(InvTemps.CLB.Decel <> InvPerms.CLB.Decel) THEN
						EPL.Param.WriteData := InvTemps.CLB.Decel;
						EPL.State := EPL_INV14_DECWRITE;
					ELSE
						EPL.State := EPL_WAIT;
						EPL.INV.DECIndex := 0;
					END_IF
				ELSE
					IF(InvPerms.CLB.Decel <> 5) THEN
						EPL.Param.WriteData := InvPerms.CLB.Decel;
						EPL.State := EPL_INV14_DECWRITE;
					ELSE
						EPL.State := EPL_INV15_ACCCHECK;
					END_IF
				END_IF
			END_IF

		EPL_INV14_DECWRITE:

			EPL.FUB.EPLWrite_0.enable := 1;  //ENABLE FUB
			EPL.FUB.EPLWrite_0.pDevice := ADR('SL1.IF1.ST17');  //DEVICE NAME OF INVERTER
			EPL.FUB.EPLWrite_0.node := 17;  //NODE NUMBER OF THE STATION
			EPL.FUB.EPLWrite_0.index := 8252;  //WRITE INDEX 16#203C (DEC 8252)
			EPL.FUB.EPLWrite_0.subindex := 3;  //SUBINDEX #2 (DEC 2) : DECELERATION RAMP
			EPL.FUB.EPLWrite_0.pData := ADR(EPL.Param.WriteData);  //POINTER TO THE DATA BEING WRITTEN
			EPL.FUB.EPLWrite_0.datalen := SIZEOF(EPL.Param.WriteData);  //SIZE OF THE DATA TO BE WRITTEN
			EPL.FUB.EPLWrite_0();

			IF EPL.FUB.EPLWrite_0.status = 0 THEN  //WRITE SUCCESSFUL
				EPL.FUB.EPLWrite_0.enable := 0;  //DISABLE THE FUB
				IF EPL.INV.DEC[14] THEN
					EPL.State := EPL_WAIT;
					EPL.INV.DECIndex := 0;
					InvPerms.CLB.Decel := InvTemps.CLB.Decel;
				ELSE
					EPL.State := EPL_INV15_ACCCHECK;
				END_IF
			ELSIF EPL.FUB.EPLWrite_0.status = ERR_FUB_BUSY THEN
				//BUSY
			ELSIF EPL.FUB.EPLWrite_0.status = ERR_FUB_ENABLE_FALSE THEN
				//DISABLED
			ELSE
				EPL.State := EPL_ERROR;
				EPL.INV.DECIndex := 0;
			END_IF

		EPL_INV15_ACCCHECK:
			EPL.State := EPL_WAIT;

		EPL_WAIT:

			FOR i := 0 TO 26 DO
				EPL.INV.ACC[i]  :=  0   ;
				EPL.INV.DEC[i]  :=  0   ;
			END_FOR

			CASE EPL.INV.ACCIndex OF
				0:
				1..26:
					EPL.INV.ACC[EPL.INV.ACCIndex] :=    TRUE    ;
					EPL.State   :=  (EPL.INV.ACCIndex * 10) ;//EPL_INV*_ACCCHECK
			END_CASE

			CASE EPL.INV.DECIndex OF
				0:
				1..26:
					EPL.INV.DEC[EPL.INV.DECIndex] :=    TRUE    ;
					EPL.State   :=  (EPL.INV.DECIndex * 10) + 2 ;//EPL_INV*_DECCHECK
			END_CASE

		EPL_ERROR:

			EPL.ErrorCode := EPL.FUB.EPLWrite_0.errorinfo;
			EPL.Status := EPL.FUB.EPLWrite_0.status;
			EPL.Errorcount := EPL.Errorcount + 1;
			EPL.State := EPL_WAIT;
			EPL.FUB.EPLWrite_0.enable := 0;

	END_CASE

END_PROGRAM
```
